// ---- DUTs/IO/PDOs/L1_Current_Status_82DECBF6.TcDUT
{attribute 'GeneratedUsingTerminal: EL3773-0000-0021'}
{attribute addProperty BoxType "EL3773-0000-0021"}
{attribute addProperty Id "I1_StatusAT %I*I1_Status_DC9039207"}
{attribute addProperty CRC "2195639286"}
{attribute addProperty Size "7"}
TYPE L1_Current_Status_82DECBF6 EXTENDS TcoIo.InputBase_8311D824 :
STRUCT
	{attribute addProperty Name "I1_Status"}
	I1_Status AT %I* : I1_Status_DC903920;
END_STRUCT
END_TYPE

// ---- DUTs/IO/PDOs/L1_Current_Samples_9EC08B3E.TcDUT
{attribute 'GeneratedUsingTerminal: EL3773-0000-0021'}
{attribute addProperty BoxType "EL3773-0000-0021"}
{attribute addProperty Id "I1_SamplesAT %I*I1_Samples_2549228720"}
{attribute addProperty CRC "2663418686"}
{attribute addProperty Size "20"}
TYPE L1_Current_Samples_9EC08B3E EXTENDS TcoIo.InputBase_8311D824 :
STRUCT
	{attribute addProperty Name "I1_Samples"}
	I1_Samples AT %I* : I1_Samples_25492287;
END_STRUCT
END_TYPE

// ---- DUTs/IO/PDOs/L2_Voltage_Status_0D1813FE.TcDUT
{attribute 'GeneratedUsingTerminal: EL3773-0000-0021'}
{attribute addProperty BoxType "EL3773-0000-0021"}
{attribute addProperty Id "U2_StatusAT %I*U2_Status_DC9039207"}
{attribute addProperty CRC "219681790"}
{attribute addProperty Size "7"}
TYPE L2_Voltage_Status_0D1813FE EXTENDS TcoIo.InputBase_8311D824 :
STRUCT
	{attribute addProperty Name "U2_Status"}
	U2_Status AT %I* : U2_Status_DC903920;
END_STRUCT
END_TYPE

// ---- DUTs/IO/PDOs/L2_Voltage_Samples_75D833AF.TcDUT
{attribute 'GeneratedUsingTerminal: EL3773-0000-0021'}
{attribute addProperty BoxType "EL3773-0000-0021"}
{attribute addProperty Id "U2_SamplesAT %I*U2_Samples_2549228720"}
{attribute addProperty CRC "1977103279"}
{attribute addProperty Size "20"}
TYPE L2_Voltage_Samples_75D833AF EXTENDS TcoIo.InputBase_8311D824 :
STRUCT
	{attribute addProperty Name "U2_Samples"}
	U2_Samples AT %I* : U2_Samples_25492287;
END_STRUCT
END_TYPE

// ---- DUTs/IO/PDOs/L2_Current_Status_FCB7684B.TcDUT
{attribute 'GeneratedUsingTerminal: EL3773-0000-0021'}
{attribute addProperty BoxType "EL3773-0000-0021"}
{attribute addProperty Id "I2_StatusAT %I*I2_Status_DC9039207"}
{attribute addProperty CRC "4239878219"}
{attribute addProperty Size "7"}
TYPE L2_Current_Status_FCB7684B EXTENDS TcoIo.InputBase_8311D824 :
STRUCT
	{attribute addProperty Name "I2_Status"}
	I2_Status AT %I* : I2_Status_DC903920;
END_STRUCT
END_TYPE

// ---- DUTs/IO/PDOs/L2_Current_Samples_AAB60F6E.TcDUT
{attribute 'GeneratedUsingTerminal: EL3773-0000-0021'}
{attribute addProperty BoxType "EL3773-0000-0021"}
{attribute addProperty Id "I2_SamplesAT %I*I2_Samples_2549228720"}
{attribute addProperty CRC "2864058222"}
{attribute addProperty Size "20"}
TYPE L2_Current_Samples_AAB60F6E EXTENDS TcoIo.InputBase_8311D824 :
STRUCT
	{attribute addProperty Name "I2_Samples"}
	I2_Samples AT %I* : I2_Samples_25492287;
END_STRUCT
END_TYPE

// ---- DUTs/IO/PDOs/L3_Voltage_Status_273F7295.TcDUT
{attribute 'GeneratedUsingTerminal: EL3773-0000-0021'}
{attribute addProperty BoxType "EL3773-0000-0021"}
{attribute addProperty Id "U3_StatusAT %I*U3_Status_DC9039207"}
{attribute addProperty CRC "658469525"}
{attribute addProperty Size "7"}
TYPE L3_Voltage_Status_273F7295 EXTENDS TcoIo.InputBase_8311D824 :
STRUCT
	{attribute addProperty Name "U3_Status"}
	U3_Status AT %I* : U3_Status_DC903920;
END_STRUCT
END_TYPE

// ---- DUTs/IO/PDOs/L3_Voltage_Samples_660A4F9F.TcDUT
{attribute 'GeneratedUsingTerminal: EL3773-0000-0021'}
{attribute addProperty BoxType "EL3773-0000-0021"}
{attribute addProperty Id "U3_SamplesAT %I*U3_Samples_2549228720"}
{attribute addProperty CRC "1711951775"}
{attribute addProperty Size "20"}
TYPE L3_Voltage_Samples_660A4F9F EXTENDS TcoIo.InputBase_8311D824 :
STRUCT
	{attribute addProperty Name "U3_Samples"}
	U3_Samples AT %I* : U3_Samples_25492287;
END_STRUCT
END_TYPE

// ---- DUTs/IO/PDOs/L3_Current_Status_D6900920.TcDUT
{attribute 'GeneratedUsingTerminal: EL3773-0000-0021'}
{attribute addProperty BoxType "EL3773-0000-0021"}
{attribute addProperty Id "I3_StatusAT %I*I3_Status_DC9039207"}
{attribute addProperty CRC "3599763744"}
{attribute addProperty Size "7"}
TYPE L3_Current_Status_D6900920 EXTENDS TcoIo.InputBase_8311D824 :
STRUCT
	{attribute addProperty Name "I3_Status"}
	I3_Status AT %I* : I3_Status_DC903920;
END_STRUCT
END_TYPE

// ---- DUTs/IO/PDOs/L3_Current_Samples_B964735E.TcDUT
{attribute 'GeneratedUsingTerminal: EL3773-0000-0021'}
{attribute addProperty BoxType "EL3773-0000-0021"}
{attribute addProperty Id "I3_SamplesAT %I*I3_Samples_2549228720"}
{attribute addProperty CRC "3110368094"}
{attribute addProperty Size "20"}
TYPE L3_Current_Samples_B964735E EXTENDS TcoIo.InputBase_8311D824 :
STRUCT
	{attribute addProperty Name "I3_Samples"}
	I3_Samples AT %I* : I3_Samples_25492287;
END_STRUCT
END_TYPE

// ---- DUTs/IO/PDOs/AI_NextSync1Time_6DC4D296.TcDUT
{attribute 'GeneratedUsingTerminal: EL3773-0000-0021'}
{attribute addProperty BoxType "EL3773-0000-0021"}
{attribute addProperty Id "StartTimeNextLatchAT %I*StartTimeNextLatch_02E0C1C88"}
{attribute addProperty CRC "1841615510"}
{attribute addProperty Size "8"}
TYPE AI_NextSync1Time_6DC4D296 EXTENDS TcoIo.InputBase_8311D824 :
STRUCT
	{attribute addProperty Name "StartTimeNextLatch"}
	StartTimeNextLatch AT %I* : StartTimeNextLatch_02E0C1C8;
END_STRUCT
END_TYPE

// ---- DUTs/IO/PDOs/AI_Sample_Count_EA88CAD9.TcDUT
{attribute 'GeneratedUsingTerminal: EL3773-0000-0021'}
{attribute addProperty BoxType "EL3773-0000-0021"}
{attribute addProperty Id "Sample_CountAT %I*UINT2"}
{attribute addProperty CRC "3934833369"}
{attribute addProperty Size "2"}
TYPE AI_Sample_Count_EA88CAD9 EXTENDS TcoIo.InputBase_8311D824 :
STRUCT
	{attribute addProperty Name "Sample_Count"}
	Sample_Count AT %I* : UINT;
END_STRUCT
END_TYPE

// ---- DUTs/IO/PDOs/InfoData_B84DBEC5.TcDUT
{attribute 'GeneratedUsingTerminal: EL3773-0000-0021'}
{attribute addProperty BoxType "EL3773-0000-0021"}
{attribute addProperty Id "AdsAddrAT %I*TcoIo.TcoAmsAddr0DcOutputShiftAT %I*DINT4DcInputShiftAT %I*DINT4StateAT %I*UINT2"}
{attribute addProperty CRC "3092102853"}
{attribute addProperty Size "10"}
TYPE InfoData_B84DBEC5 EXTENDS TcoIo.InputBase_8311D824 :
STRUCT
	{attribute addProperty Name "AdsAddr"}
	AdsAddr AT %I* : TcoIo.TcoAmsAddr;
	{attribute addProperty Name "DcOutputShift"}
	DcOutputShift AT %I* : DINT;
	{attribute addProperty Name "DcInputShift"}
	DcInputShift AT %I* : DINT;
	{attribute addProperty Name "State"}
	State AT %I* : UINT;
END_STRUCT
END_TYPE

// ---- DUTs/IO/PDOs/MTO_Inputs_Channel_53C09E8B.TcDUT
{attribute 'GeneratedUsingTerminal: EL2258-0000-0017'}
{attribute addProperty BoxType "EL2258-0000-0017"}
{attribute addProperty Id "StatusAT %I*Status_642C2ED16"}
{attribute addProperty CRC "1405132427"}
{attribute addProperty Size "6"}
TYPE MTO_Inputs_Channel_53C09E8B EXTENDS TcoIo.InputBase_8311D824 :
STRUCT
	{attribute addProperty Name "Status"}
	Status AT %I* : Status_642C2ED1;
END_STRUCT
END_TYPE

// ---- DUTs/IO/PDOs/MTO_Outputs_10x_Channel_A3C0C022.TcDUT
{attribute 'GeneratedUsingTerminal: EL2258-0000-0017'}
{attribute addProperty BoxType "EL2258-0000-0017"}
{attribute addProperty Id "CtrlAT %Q*Ctrl_77460BD36OutputsAT %Q*Outputs_A910484D10Output_event_timeAT %Q*ARRAY[0..9] OF UDINT40"}
{attribute addProperty CRC "922776817"}
{attribute addProperty Size "56"}
TYPE MTO_Outputs_10x_Channel_A3C0C022 EXTENDS TcoIo.OutputBase_10CEE7DE :
STRUCT
	{attribute addProperty Name "Ctrl"}
	Ctrl AT %Q* : Ctrl_77460BD3;
	{attribute addProperty Name "Outputs"}
	Outputs AT %Q* : Outputs_A910484D;
	{attribute addProperty Name "Output_event_time"}
	Output_event_time AT %Q* : ARRAY[0..9] OF UDINT;
END_STRUCT
END_TYPE

// ---- DUTs/IO/PDOs/PM_Inputs_Channel_2F868086.TcDUT
{attribute 'GeneratedUsingTerminal: EL3403-0000-0023'}
{attribute addProperty BoxType "EL3403-0000-0023"}
{attribute addProperty Id "TxPDO_ToggleAT %I*BOOL1CurrentAT %I*DINT4VoltageAT %I*DINT4Active_powerAT %I*DINT4IndexAT %I*USINT1Variant_valueAT %I*DINT4"}
{attribute addProperty CRC "797343878"}
{attribute addProperty Size "18"}
TYPE PM_Inputs_Channel_2F868086 EXTENDS TcoIo.InputBase_8311D824 :
STRUCT
	{attribute addProperty Name "TxPDO_Toggle"}
	TxPDO_Toggle AT %I* : BOOL;
	{attribute addProperty Name "Current"}
	Current AT %I* : DINT;
	{attribute addProperty Name "Voltage"}
	Voltage AT %I* : DINT;
	{attribute addProperty Name "Active_power"}
	Active_power AT %I* : DINT;
	{attribute addProperty Name "Index"}
	Index AT %I* : USINT;
	{attribute addProperty Name "Variant_value"}
	Variant_value AT %I* : DINT;
END_STRUCT
END_TYPE

// ---- DUTs/IO/PDOs/PM_Status_data_2A9514CB.TcDUT
{attribute 'GeneratedUsingTerminal: EL3403-0000-0023'}
{attribute addProperty BoxType "EL3403-0000-0023"}
{attribute addProperty Id "Missing_zero_crossing_AAT %I*BOOL1Missing_zero_crossing_BAT %I*BOOL1Missing_zero_crossing_CAT %I*BOOL1Phase_sequence_errorAT %I*BOOL1"}
{attribute addProperty CRC "714413259"}
{attribute addProperty Size "4"}
TYPE PM_Status_data_2A9514CB EXTENDS TcoIo.InputBase_8311D824 :
STRUCT
	{attribute addProperty Name "Missing_zero_crossing_A"}
	Missing_zero_crossing_A AT %I* : BOOL;
	{attribute addProperty Name "Missing_zero_crossing_B"}
	Missing_zero_crossing_B AT %I* : BOOL;
	{attribute addProperty Name "Missing_zero_crossing_C"}
	Missing_zero_crossing_C AT %I* : BOOL;
	{attribute addProperty Name "Phase_sequence_error"}
	Phase_sequence_error AT %I* : BOOL;
END_STRUCT
END_TYPE

// ---- DUTs/IO/PDOs/PM_Outputs_Channel_E5FBDE30.TcDUT
{attribute 'GeneratedUsingTerminal: EL3403-0000-0023'}
{attribute addProperty BoxType "EL3403-0000-0023"}
{attribute addProperty Id "IndexAT %Q*USINT1"}
{attribute addProperty CRC "3858488880"}
{attribute addProperty Size "1"}
TYPE PM_Outputs_Channel_E5FBDE30 EXTENDS TcoIo.OutputBase_10CEE7DE :
STRUCT
	{attribute addProperty Name "Index"}
	Index AT %Q* : USINT;
END_STRUCT
END_TYPE

// ---- DUTs/IO/PDOs/AT_x_4EC2E768.TcDUT
{attribute 'GeneratedUsingTerminal: AX5101-0000-0214-0214'}
{attribute addProperty BoxType "AX5101-0000-0214-0214"}
{attribute addProperty Id "Drive_status_wordAT %I*UINT2Position_feedback_1_valueAT %I*DINT4Following_distanceAT %I*DINT4"}
{attribute addProperty CRC "1321396072"}
{attribute addProperty Size "10"}
TYPE AT_x_4EC2E768 EXTENDS TcoIo.InputBase_8311D824 :
STRUCT
	{attribute addProperty Name "Drive_status_word"}
	Drive_status_word AT %I* : UINT;
	{attribute addProperty Name "Position_feedback_1_value"}
	Position_feedback_1_value AT %I* : DINT;
	{attribute addProperty Name "Following_distance"}
	Following_distance AT %I* : DINT;
END_STRUCT
END_TYPE

// ---- DUTs/IO/PDOs/MDT_864618EC.TcDUT
{attribute 'GeneratedUsingTerminal: AX5101-0000-0214-0214'}
{attribute addProperty BoxType "AX5101-0000-0214-0214"}
{attribute addProperty Id "Master_control_wordAT %Q*UINT2Position_command_valueAT %Q*DINT4"}
{attribute addProperty CRC "2252740844"}
{attribute addProperty Size "6"}
TYPE MDT_864618EC EXTENDS TcoIo.OutputBase_10CEE7DE :
STRUCT
	{attribute addProperty Name "Master_control_word"}
	Master_control_word AT %Q* : UINT;
	{attribute addProperty Name "Position_command_value"}
	Position_command_value AT %Q* : DINT;
END_STRUCT
END_TYPE

// ---- DUTs/IO/PDOs/InfoData_F60A43AC.TcDUT
{attribute 'GeneratedUsingTerminal: AX5101-0000-0214-0214'}
{attribute addProperty BoxType "AX5101-0000-0214-0214"}
{attribute addProperty Id "AdsAddrAT %I*TcoIo.TcoAmsAddr0DcOutputShiftAT %I*DINT4DcInputShiftAT %I*DINT4Chn0AT %I*USINT1StateAT %I*UINT2"}
{attribute addProperty CRC "4127867820"}
{attribute addProperty Size "11"}
TYPE InfoData_F60A43AC EXTENDS TcoIo.InputBase_8311D824 :
STRUCT
	{attribute addProperty Name "AdsAddr"}
	AdsAddr AT %I* : TcoIo.TcoAmsAddr;
	{attribute addProperty Name "DcOutputShift"}
	DcOutputShift AT %I* : DINT;
	{attribute addProperty Name "DcInputShift"}
	DcInputShift AT %I* : DINT;
	{attribute addProperty Name "Chn0"}
	Chn0 AT %I* : USINT;
	{attribute addProperty Name "State"}
	State AT %I* : UINT;
END_STRUCT
END_TYPE

// ---- DUTs/IO/Boxes/EK1200_013D0B49.TcDUT
{attribute 'GeneratedUsingTerminal: EK1200-1388-0000'}
{attribute addProperty VendorId "#x00000002"}
{attribute addProperty BoxType "EK1200-1388-0000"}
{attribute addProperty Description "EK1200-5000 EtherCAT Power supply (2A E-Bus)"}
{attribute addProperty Physics "YK"}
{attribute addProperty Id "EK1200"}
{attribute addProperty CRC "20777801"}
{attribute addProperty Size "0"}
TYPE EK1200_013D0B49 EXTENDS TcoIo.EtcSlaveBoxBase_77A0E4A7 :
STRUCT
END_STRUCT
END_TYPE

// ---- DUTs/IO/Boxes/EL6002_CD897635.TcDUT
{attribute 'GeneratedUsingTerminal: EL6002-0000-0019'}
{attribute addProperty VendorId "#x00000002"}
{attribute addProperty BoxType "EL6002-0000-0019"}
{attribute addProperty Description "EL6002 Interface 2Ch. (RS232)"}
{attribute addProperty Physics "KK"}
{attribute addProperty Id "COM_TxPDO_Map_Inputs_Channel_1AT %I*COM_TxPDO_Map_Inputs_Channel_3801C95E30COM_TxPDO_Map_Inputs_Channel_2AT %I*COM_TxPDO_Map_Inputs_Channel_3801C95E30COM_RxPDO_Map_Outputs_Channel_1AT %Q*COM_RxPDO_Map_Outputs_Channel_EADA2E0D27COM_RxPDO_Map_Outputs_Channel_2AT %Q*COM_RxPDO_Map_Outputs_Channel_EADA2E0D27WcStateAT %I*WcState_9091E0EB2InfoDataAT %I*InfoData_23CBA8372"}
{attribute addProperty CRC "3448337973"}
{attribute addProperty Size "118"}
TYPE EL6002_CD897635 EXTENDS TcoIo.EtcSlaveTerminalBase_947E5A46 :
STRUCT
	{attribute addProperty Name "COM_TxPDO_Map_Inputs_Channel_1"}
	COM_TxPDO_Map_Inputs_Channel_1 : COM_TxPDO_Map_Inputs_Channel_3801C95E;
	{attribute addProperty Name "COM_TxPDO_Map_Inputs_Channel_2"}
	COM_TxPDO_Map_Inputs_Channel_2 : COM_TxPDO_Map_Inputs_Channel_3801C95E;
	{attribute addProperty Name "COM_RxPDO_Map_Outputs_Channel_1"}
	COM_RxPDO_Map_Outputs_Channel_1 : COM_RxPDO_Map_Outputs_Channel_EADA2E0D;
	{attribute addProperty Name "COM_RxPDO_Map_Outputs_Channel_2"}
	COM_RxPDO_Map_Outputs_Channel_2 : COM_RxPDO_Map_Outputs_Channel_EADA2E0D;
	{attribute addProperty Name "WcState"}
	WcState : TcoIo.WcState_9091E0EB;
	{attribute addProperty Name "InfoData"}
	InfoData : TcoIo.InfoData_23CBA837;
END_STRUCT
END_TYPE

// ---- DUTs/IO/Boxes/EL1809_32157CFD.TcDUT
{attribute 'GeneratedUsingTerminal: EL1809-0000-0018'}
{attribute addProperty VendorId "#x00000002"}
{attribute addProperty BoxType "EL1809-0000-0018"}
{attribute addProperty Description "EL1809 16Ch. Dig. Input 24V, 3ms"}
{attribute addProperty Physics "KK"}
{attribute addProperty Id "Channel_1AT %I*Channel_830843C11Channel_2AT %I*Channel_830843C11Channel_3AT %I*Channel_830843C11Channel_4AT %I*Channel_830843C11Channel_5AT %I*Channel_830843C11Channel_6AT %I*Channel_830843C11Channel_7AT %I*Channel_830843C11Channel_8AT %I*Channel_830843C11Channel_9AT %I*Channel_830843C11Channel_10AT %I*Channel_830843C11Channel_11AT %I*Channel_830843C11Channel_12AT %I*Channel_830843C11Channel_13AT %I*Channel_830843C11Channel_14AT %I*Channel_830843C11Channel_15AT %I*Channel_830843C11Channel_16AT %I*Channel_830843C11WcStateAT %I*WcState_9091E0EB2InfoDataAT %I*InfoData_6F19DB2B2"}
{attribute addProperty CRC "840269053"}
{attribute addProperty Size "20"}
TYPE EL1809_32157CFD EXTENDS TcoIo.EtcSlaveTerminalBase_947E5A46 :
STRUCT
	{attribute addProperty Name "Channel_1"}
	Channel_1 : Channel_830843C1;
	{attribute addProperty Name "Channel_2"}
	Channel_2 : Channel_830843C1;
	{attribute addProperty Name "Channel_3"}
	Channel_3 : Channel_830843C1;
	{attribute addProperty Name "Channel_4"}
	Channel_4 : Channel_830843C1;
	{attribute addProperty Name "Channel_5"}
	Channel_5 : Channel_830843C1;
	{attribute addProperty Name "Channel_6"}
	Channel_6 : Channel_830843C1;
	{attribute addProperty Name "Channel_7"}
	Channel_7 : Channel_830843C1;
	{attribute addProperty Name "Channel_8"}
	Channel_8 : Channel_830843C1;
	{attribute addProperty Name "Channel_9"}
	Channel_9 : Channel_830843C1;
	{attribute addProperty Name "Channel_10"}
	Channel_10 : Channel_830843C1;
	{attribute addProperty Name "Channel_11"}
	Channel_11 : Channel_830843C1;
	{attribute addProperty Name "Channel_12"}
	Channel_12 : Channel_830843C1;
	{attribute addProperty Name "Channel_13"}
	Channel_13 : Channel_830843C1;
	{attribute addProperty Name "Channel_14"}
	Channel_14 : Channel_830843C1;
	{attribute addProperty Name "Channel_15"}
	Channel_15 : Channel_830843C1;
	{attribute addProperty Name "Channel_16"}
	Channel_16 : Channel_830843C1;
	{attribute addProperty Name "WcState"}
	WcState : TcoIo.WcState_9091E0EB;
	{attribute addProperty Name "InfoData"}
	InfoData : TcoIo.InfoData_6F19DB2B;
END_STRUCT
END_TYPE

// ---- DUTs/IO/Boxes/EL2809_2B6483BD.TcDUT
{attribute 'GeneratedUsingTerminal: EL2809-0000-0018'}
{attribute addProperty VendorId "#x00000002"}
{attribute addProperty BoxType "EL2809-0000-0018"}
{attribute addProperty Description "EL2809 16Ch. Dig. Output 24V, 0.5A"}
{attribute addProperty Physics "KK"}
{attribute addProperty Id "Channel_1AT %Q*Channel_42CA91F71Channel_2AT %Q*Channel_42CA91F71Channel_3AT %Q*Channel_42CA91F71Channel_4AT %Q*Channel_42CA91F71Channel_5AT %Q*Channel_42CA91F71Channel_6AT %Q*Channel_42CA91F71Channel_7AT %Q*Channel_42CA91F71Channel_8AT %Q*Channel_42CA91F71Channel_9AT %Q*Channel_42CA91F71Channel_10AT %Q*Channel_42CA91F71Channel_11AT %Q*Channel_42CA91F71Channel_12AT %Q*Channel_42CA91F71Channel_13AT %Q*Channel_42CA91F71Channel_14AT %Q*Channel_42CA91F71Channel_15AT %Q*Channel_42CA91F71Channel_16AT %Q*Channel_42CA91F71WcStateAT %I*WcState_0B2B16F91InfoDataAT %I*InfoData_6F19DB2B2"}
{attribute addProperty CRC "728007613"}
{attribute addProperty Size "19"}
TYPE EL2809_2B6483BD EXTENDS TcoIo.EtcSlaveTerminalBase_947E5A46 :
STRUCT
	{attribute addProperty Name "Channel_1"}
	Channel_1 : Channel_42CA91F7;
	{attribute addProperty Name "Channel_2"}
	Channel_2 : Channel_42CA91F7;
	{attribute addProperty Name "Channel_3"}
	Channel_3 : Channel_42CA91F7;
	{attribute addProperty Name "Channel_4"}
	Channel_4 : Channel_42CA91F7;
	{attribute addProperty Name "Channel_5"}
	Channel_5 : Channel_42CA91F7;
	{attribute addProperty Name "Channel_6"}
	Channel_6 : Channel_42CA91F7;
	{attribute addProperty Name "Channel_7"}
	Channel_7 : Channel_42CA91F7;
	{attribute addProperty Name "Channel_8"}
	Channel_8 : Channel_42CA91F7;
	{attribute addProperty Name "Channel_9"}
	Channel_9 : Channel_42CA91F7;
	{attribute addProperty Name "Channel_10"}
	Channel_10 : Channel_42CA91F7;
	{attribute addProperty Name "Channel_11"}
	Channel_11 : Channel_42CA91F7;
	{attribute addProperty Name "Channel_12"}
	Channel_12 : Channel_42CA91F7;
	{attribute addProperty Name "Channel_13"}
	Channel_13 : Channel_42CA91F7;
	{attribute addProperty Name "Channel_14"}
	Channel_14 : Channel_42CA91F7;
	{attribute addProperty Name "Channel_15"}
	Channel_15 : Channel_42CA91F7;
	{attribute addProperty Name "Channel_16"}
	Channel_16 : Channel_42CA91F7;
	{attribute addProperty Name "WcState"}
	WcState : TcoIo.WcState_0B2B16F9;
	{attribute addProperty Name "InfoData"}
	InfoData : TcoIo.InfoData_6F19DB2B;
END_STRUCT
END_TYPE

// ---- DUTs/IO/Boxes/EL4004_E203F875.TcDUT
{attribute 'GeneratedUsingTerminal: EL4004-0000-0020'}
{attribute addProperty VendorId "#x00000002"}
{attribute addProperty BoxType "EL4004-0000-0020"}
{attribute addProperty Description "EL4004 4Ch. Ana. Output 0-10V, 12bit"}
{attribute addProperty Physics "KK"}
{attribute addProperty Id "AO_Outputs_Channel_1AT %Q*AO_Output_Channel_BA7EBB7C2AO_Outputs_Channel_2AT %Q*AO_Output_Channel_BA7EBB7C2AO_Outputs_Channel_3AT %Q*AO_Output_Channel_BA7EBB7C2AO_Outputs_Channel_4AT %Q*AO_Output_Channel_BA7EBB7C2WcStateAT %I*WcState_0B2B16F91InfoDataAT %I*InfoData_23CBA8372"}
{attribute addProperty CRC "3791911029"}
{attribute addProperty Size "11"}
TYPE EL4004_E203F875 EXTENDS TcoIo.EtcSlaveTerminalBase_947E5A46 :
STRUCT
	{attribute addProperty Name "AO_Outputs_Channel_1"}
	AO_Outputs_Channel_1 : AO_Output_Channel_BA7EBB7C;
	{attribute addProperty Name "AO_Outputs_Channel_2"}
	AO_Outputs_Channel_2 : AO_Output_Channel_BA7EBB7C;
	{attribute addProperty Name "AO_Outputs_Channel_3"}
	AO_Outputs_Channel_3 : AO_Output_Channel_BA7EBB7C;
	{attribute addProperty Name "AO_Outputs_Channel_4"}
	AO_Outputs_Channel_4 : AO_Output_Channel_BA7EBB7C;
	{attribute addProperty Name "WcState"}
	WcState : TcoIo.WcState_0B2B16F9;
	{attribute addProperty Name "InfoData"}
	InfoData : TcoIo.InfoData_23CBA837;
END_STRUCT
END_TYPE

// ---- DUTs/IO/Boxes/EL6001_0DE01E7E.TcDUT
{attribute 'GeneratedUsingTerminal: EL6001-0000-0020'}
{attribute addProperty VendorId "#x00000002"}
{attribute addProperty BoxType "EL6001-0000-0020"}
{attribute addProperty Description "EL6001 Interface (RS232)"}
{attribute addProperty Physics "KK"}
{attribute addProperty Id "COM_InputsAT %I*COM_Inputs_3801C95E30COM_OutputsAT %Q*COM_Outputs_DEF408EC27WcStateAT %I*WcState_9091E0EB2InfoDataAT %I*InfoData_23CBA8372"}
{attribute addProperty CRC "232791678"}
{attribute addProperty Size "61"}
TYPE EL6001_0DE01E7E EXTENDS TcoIo.EtcSlaveTerminalBase_947E5A46 :
STRUCT
	{attribute addProperty Name "COM_Inputs"}
	COM_Inputs : COM_Inputs_3801C95E;
	{attribute addProperty Name "COM_Outputs"}
	COM_Outputs : COM_Outputs_DEF408EC;
	{attribute addProperty Name "WcState"}
	WcState : TcoIo.WcState_9091E0EB;
	{attribute addProperty Name "InfoData"}
	InfoData : TcoIo.InfoData_23CBA837;
END_STRUCT
END_TYPE

// ---- DUTs/IO/Boxes/EL9011_D65D3D32.TcDUT
{attribute 'GeneratedUsingTerminal: EL9011--0000'}
{attribute addProperty VendorId "#x00000002"}
{attribute addProperty BoxType "EL9011--0000"}
{attribute addProperty Description "EL9011 End Terminal"}
{attribute addProperty Physics ""}
{attribute addProperty Id "EL9011"}
{attribute addProperty CRC "3596434738"}
{attribute addProperty Size "0"}
TYPE EL9011_D65D3D32 EXTENDS TcoIo.EtcSlaveEndTerminalBase_866C7F0C :
STRUCT
END_STRUCT
END_TYPE

// ---- DUTs/IO/Boxes/EK1100_1FC0878B.TcDUT
{attribute 'GeneratedUsingTerminal: EK1100-0000-0018'}
{attribute addProperty VendorId "#x00000002"}
{attribute addProperty BoxType "EK1100-0000-0018"}
{attribute addProperty Description "EK1100 EtherCAT Coupler (2A E-Bus)"}
{attribute addProperty Physics "YKY"}
{attribute addProperty Id "InfoDataAT %I*InfoData_6F19DB2B2"}
{attribute addProperty CRC "532711307"}
{attribute addProperty Size "2"}
TYPE EK1100_1FC0878B EXTENDS TcoIo.EtcSlaveBoxBase_77A0E4A7 :
STRUCT
	{attribute addProperty Name "InfoData"}
	InfoData : TcoIo.InfoData_6F19DB2B;
END_STRUCT
END_TYPE

// ---- DUTs/IO/Boxes/EK1122_1FC0878B.TcDUT
{attribute 'GeneratedUsingTerminal: EK1122-0000-0018'}
{attribute addProperty VendorId "#x00000002"}
{attribute addProperty BoxType "EK1122-0000-0018"}
{attribute addProperty Description "EK1122 2 port EtherCAT junction"}
{attribute addProperty Physics "KYKY"}
{attribute addProperty Id "InfoDataAT %I*InfoData_6F19DB2B2"}
{attribute addProperty CRC "532711307"}
{attribute addProperty Size "2"}
TYPE EK1122_1FC0878B EXTENDS TcoIo.EtcSlaveTerminalBase_947E5A46 :
STRUCT
	{attribute addProperty Name "InfoData"}
	InfoData : TcoIo.InfoData_6F19DB2B;
END_STRUCT
END_TYPE

// ---- DUTs/IO/Boxes/EL3174_B71BFF42.TcDUT
{attribute 'GeneratedUsingTerminal: EL3174-0002-0017'}
{attribute addProperty VendorId "#x00000002"}
{attribute addProperty BoxType "EL3174-0002-0017"}
{attribute addProperty Description "EL3174-0002 4Ch. Ana. Input +/-10V, +/-20mA 16 Bit, Isolated Channels"}
{attribute addProperty Physics "KK"}
{attribute addProperty Id "AI_Standard_Channel_1AT %I*AI_Standard_Channel_A8DF64E310AI_Standard_Channel_2AT %I*AI_Standard_Channel_A8DF64E310AI_Standard_Channel_3AT %I*AI_Standard_Channel_A8DF64E310AI_Standard_Channel_4AT %I*AI_Standard_Channel_A8DF64E310WcStateAT %I*WcState_9091E0EB2InfoDataAT %I*InfoData_23CBA8372"}
{attribute addProperty CRC "3072065346"}
{attribute addProperty Size "44"}
TYPE EL3174_B71BFF42 EXTENDS TcoIo.EtcSlaveTerminalBase_947E5A46 :
STRUCT
	{attribute addProperty Name "AI_Standard_Channel_1"}
	AI_Standard_Channel_1 : AI_Standard_Channel_A8DF64E3;
	{attribute addProperty Name "AI_Standard_Channel_2"}
	AI_Standard_Channel_2 : AI_Standard_Channel_A8DF64E3;
	{attribute addProperty Name "AI_Standard_Channel_3"}
	AI_Standard_Channel_3 : AI_Standard_Channel_A8DF64E3;
	{attribute addProperty Name "AI_Standard_Channel_4"}
	AI_Standard_Channel_4 : AI_Standard_Channel_A8DF64E3;
	{attribute addProperty Name "WcState"}
	WcState : TcoIo.WcState_9091E0EB;
	{attribute addProperty Name "InfoData"}
	InfoData : TcoIo.InfoData_23CBA837;
END_STRUCT
END_TYPE

// ---- DUTs/IO/Boxes/EL3011_7A495228.TcDUT
{attribute 'GeneratedUsingTerminal: EL3011-0000-0018'}
{attribute addProperty VendorId "#x00000002"}
{attribute addProperty BoxType "EL3011-0000-0018"}
{attribute addProperty Description "EL3011 4Ch. Ana. Input 0-20mA DIFF"}
{attribute addProperty Physics "KK"}
{attribute addProperty Id "AI_StandardAT %I*AI_Standard_Channel_4A3944819WcStateAT %I*WcState_9091E0EB2InfoDataAT %I*InfoData_23CBA8372"}
{attribute addProperty CRC "2051625512"}
{attribute addProperty Size "13"}
TYPE EL3011_7A495228 EXTENDS TcoIo.EtcSlaveTerminalBase_947E5A46 :
STRUCT
	{attribute addProperty Name "AI_Standard"}
	AI_Standard : AI_Standard_Channel_4A394481;
	{attribute addProperty Name "WcState"}
	WcState : TcoIo.WcState_9091E0EB;
	{attribute addProperty Name "InfoData"}
	InfoData : TcoIo.InfoData_23CBA837;
END_STRUCT
END_TYPE

// ---- DUTs/IO/Boxes/EL2008_E2806B95.TcDUT
{attribute 'GeneratedUsingTerminal: EL2008-0000-0017'}
{attribute addProperty VendorId "#x00000002"}
{attribute addProperty BoxType "EL2008-0000-0017"}
{attribute addProperty Description "EL2008 8Ch. Dig. Output 24V, 0.5A"}
{attribute addProperty Physics "KK"}
{attribute addProperty Id "Channel_1AT %Q*Channel_42CA91F71Channel_2AT %Q*Channel_42CA91F71Channel_3AT %Q*Channel_42CA91F71Channel_4AT %Q*Channel_42CA91F71Channel_5AT %Q*Channel_42CA91F71Channel_6AT %Q*Channel_42CA91F71Channel_7AT %Q*Channel_42CA91F71Channel_8AT %Q*Channel_42CA91F71WcStateAT %I*WcState_0B2B16F91InfoDataAT %I*InfoData_6F19DB2B2"}
{attribute addProperty CRC "3800066965"}
{attribute addProperty Size "11"}
TYPE EL2008_E2806B95 EXTENDS TcoIo.EtcSlaveTerminalBase_947E5A46 :
STRUCT
	{attribute addProperty Name "Channel_1"}
	Channel_1 : Channel_42CA91F7;
	{attribute addProperty Name "Channel_2"}
	Channel_2 : Channel_42CA91F7;
	{attribute addProperty Name "Channel_3"}
	Channel_3 : Channel_42CA91F7;
	{attribute addProperty Name "Channel_4"}
	Channel_4 : Channel_42CA91F7;
	{attribute addProperty Name "Channel_5"}
	Channel_5 : Channel_42CA91F7;
	{attribute addProperty Name "Channel_6"}
	Channel_6 : Channel_42CA91F7;
	{attribute addProperty Name "Channel_7"}
	Channel_7 : Channel_42CA91F7;
	{attribute addProperty Name "Channel_8"}
	Channel_8 : Channel_42CA91F7;
	{attribute addProperty Name "WcState"}
	WcState : TcoIo.WcState_0B2B16F9;
	{attribute addProperty Name "InfoData"}
	InfoData : TcoIo.InfoData_6F19DB2B;
END_STRUCT
END_TYPE

// ---- DUTs/IO/Boxes/EK1110_1FC0878B.TcDUT
{attribute 'GeneratedUsingTerminal: EK1110-0000-0017'}
{attribute addProperty VendorId "#x00000002"}
{attribute addProperty BoxType "EK1110-0000-0017"}
{attribute addProperty Description "EK1110 EtherCAT extension"}
{attribute addProperty Physics "KY"}
{attribute addProperty Id "InfoDataAT %I*InfoData_6F19DB2B2"}
{attribute addProperty CRC "532711307"}
{attribute addProperty Size "2"}
TYPE EK1110_1FC0878B EXTENDS TcoIo.EtcSlaveTerminalBase_947E5A46 :
STRUCT
	{attribute addProperty Name "InfoData"}
	InfoData : TcoIo.InfoData_6F19DB2B;
END_STRUCT
END_TYPE

// ---- DUTs/IO/Boxes/EL1819_32157CFD.TcDUT
{attribute 'GeneratedUsingTerminal: EL1819-0000-0018'}
{attribute addProperty VendorId "#x00000002"}
{attribute addProperty BoxType "EL1819-0000-0018"}
{attribute addProperty Description "EL1819 16Ch. Dig. Input 24V, 10Ã‚Âµs"}
{attribute addProperty Physics "KK"}
{attribute addProperty Id "Channel_1AT %I*Channel_830843C11Channel_2AT %I*Channel_830843C11Channel_3AT %I*Channel_830843C11Channel_4AT %I*Channel_830843C11Channel_5AT %I*Channel_830843C11Channel_6AT %I*Channel_830843C11Channel_7AT %I*Channel_830843C11Channel_8AT %I*Channel_830843C11Channel_9AT %I*Channel_830843C11Channel_10AT %I*Channel_830843C11Channel_11AT %I*Channel_830843C11Channel_12AT %I*Channel_830843C11Channel_13AT %I*Channel_830843C11Channel_14AT %I*Channel_830843C11Channel_15AT %I*Channel_830843C11Channel_16AT %I*Channel_830843C11WcStateAT %I*WcState_9091E0EB2InfoDataAT %I*InfoData_6F19DB2B2"}
{attribute addProperty CRC "840269053"}
{attribute addProperty Size "20"}
TYPE EL1819_32157CFD EXTENDS TcoIo.EtcSlaveTerminalBase_947E5A46 :
STRUCT
	{attribute addProperty Name "Channel_1"}
	Channel_1 : Channel_830843C1;
	{attribute addProperty Name "Channel_2"}
	Channel_2 : Channel_830843C1;
	{attribute addProperty Name "Channel_3"}
	Channel_3 : Channel_830843C1;
	{attribute addProperty Name "Channel_4"}
	Channel_4 : Channel_830843C1;
	{attribute addProperty Name "Channel_5"}
	Channel_5 : Channel_830843C1;
	{attribute addProperty Name "Channel_6"}
	Channel_6 : Channel_830843C1;
	{attribute addProperty Name "Channel_7"}
	Channel_7 : Channel_830843C1;
	{attribute addProperty Name "Channel_8"}
	Channel_8 : Channel_830843C1;
	{attribute addProperty Name "Channel_9"}
	Channel_9 : Channel_830843C1;
	{attribute addProperty Name "Channel_10"}
	Channel_10 : Channel_830843C1;
	{attribute addProperty Name "Channel_11"}
	Channel_11 : Channel_830843C1;
	{attribute addProperty Name "Channel_12"}
	Channel_12 : Channel_830843C1;
	{attribute addProperty Name "Channel_13"}
	Channel_13 : Channel_830843C1;
	{attribute addProperty Name "Channel_14"}
	Channel_14 : Channel_830843C1;
	{attribute addProperty Name "Channel_15"}
	Channel_15 : Channel_830843C1;
	{attribute addProperty Name "Channel_16"}
	Channel_16 : Channel_830843C1;
	{attribute addProperty Name "WcState"}
	WcState : TcoIo.WcState_9091E0EB;
	{attribute addProperty Name "InfoData"}
	InfoData : TcoIo.InfoData_6F19DB2B;
END_STRUCT
END_TYPE

// ---- DUTs/IO/Boxes/EL2788_E2806B95.TcDUT
{attribute 'GeneratedUsingTerminal: EL2788-0000-0016'}
{attribute addProperty VendorId "#x00000002"}
{attribute addProperty BoxType "EL2788-0000-0016"}
{attribute addProperty Description "EL2788 8Ch. Dig. Output 24V AC/DC, 2A"}
{attribute addProperty Physics "KK"}
{attribute addProperty Id "Channel_1AT %Q*Channel_42CA91F71Channel_2AT %Q*Channel_42CA91F71Channel_3AT %Q*Channel_42CA91F71Channel_4AT %Q*Channel_42CA91F71Channel_5AT %Q*Channel_42CA91F71Channel_6AT %Q*Channel_42CA91F71Channel_7AT %Q*Channel_42CA91F71Channel_8AT %Q*Channel_42CA91F71WcStateAT %I*WcState_0B2B16F91InfoDataAT %I*InfoData_6F19DB2B2"}
{attribute addProperty CRC "3800066965"}
{attribute addProperty Size "11"}
TYPE EL2788_E2806B95 EXTENDS TcoIo.EtcSlaveTerminalBase_947E5A46 :
STRUCT
	{attribute addProperty Name "Channel_1"}
	Channel_1 : Channel_42CA91F7;
	{attribute addProperty Name "Channel_2"}
	Channel_2 : Channel_42CA91F7;
	{attribute addProperty Name "Channel_3"}
	Channel_3 : Channel_42CA91F7;
	{attribute addProperty Name "Channel_4"}
	Channel_4 : Channel_42CA91F7;
	{attribute addProperty Name "Channel_5"}
	Channel_5 : Channel_42CA91F7;
	{attribute addProperty Name "Channel_6"}
	Channel_6 : Channel_42CA91F7;
	{attribute addProperty Name "Channel_7"}
	Channel_7 : Channel_42CA91F7;
	{attribute addProperty Name "Channel_8"}
	Channel_8 : Channel_42CA91F7;
	{attribute addProperty Name "WcState"}
	WcState : TcoIo.WcState_0B2B16F9;
	{attribute addProperty Name "InfoData"}
	InfoData : TcoIo.InfoData_6F19DB2B;
END_STRUCT
END_TYPE

// ---- DUTs/IO/Boxes/EL3773_F128CC82.TcDUT
{attribute 'GeneratedUsingTerminal: EL3773-0000-0021'}
{attribute addProperty VendorId "#x00000002"}
{attribute addProperty BoxType "EL3773-0000-0021"}
{attribute addProperty Description "EL3773 3 Ch. Power Monitoring, Oversample"}
{attribute addProperty Physics "KK"}
{attribute addProperty Id "L1_Voltage_StatusAT %I*L1_Voltage_Status_7371B0437L1_Voltage_SamplesAT %I*L1_Voltage_Samples_41AEB7FF20L1_Current_StatusAT %I*L1_Current_Status_82DECBF67L1_Current_SamplesAT %I*L1_Current_Samples_9EC08B3E20L2_Voltage_StatusAT %I*L2_Voltage_Status_0D1813FE7L2_Voltage_SamplesAT %I*L2_Voltage_Samples_75D833AF20L2_Current_StatusAT %I*L2_Current_Status_FCB7684B7L2_Current_SamplesAT %I*L2_Current_Samples_AAB60F6E20L3_Voltage_StatusAT %I*L3_Voltage_Status_273F72957L3_Voltage_SamplesAT %I*L3_Voltage_Samples_660A4F9F20L3_Current_StatusAT %I*L3_Current_Status_D69009207L3_Current_SamplesAT %I*L3_Current_Samples_B964735E20AI_NextSync1TimeAT %I*AI_NextSync1Time_6DC4D2968AI_Sample_CountAT %I*AI_Sample_Count_EA88CAD92WcStateAT %I*WcState_9091E0EB2InfoDataAT %I*InfoData_B84DBEC510"}
{attribute addProperty CRC "4045982850"}
{attribute addProperty Size "184"}
TYPE EL3773_F128CC82 EXTENDS TcoIo.EtcSlaveTerminalBase_947E5A46 :
STRUCT
	{attribute addProperty Name "L1_Voltage_Status"}
	L1_Voltage_Status : L1_Voltage_Status_7371B043;
	{attribute addProperty Name "L1_Voltage_Samples"}
	L1_Voltage_Samples : L1_Voltage_Samples_41AEB7FF;
	{attribute addProperty Name "L1_Current_Status"}
	L1_Current_Status : L1_Current_Status_82DECBF6;
	{attribute addProperty Name "L1_Current_Samples"}
	L1_Current_Samples : L1_Current_Samples_9EC08B3E;
	{attribute addProperty Name "L2_Voltage_Status"}
	L2_Voltage_Status : L2_Voltage_Status_0D1813FE;
	{attribute addProperty Name "L2_Voltage_Samples"}
	L2_Voltage_Samples : L2_Voltage_Samples_75D833AF;
	{attribute addProperty Name "L2_Current_Status"}
	L2_Current_Status : L2_Current_Status_FCB7684B;
	{attribute addProperty Name "L2_Current_Samples"}
	L2_Current_Samples : L2_Current_Samples_AAB60F6E;
	{attribute addProperty Name "L3_Voltage_Status"}
	L3_Voltage_Status : L3_Voltage_Status_273F7295;
	{attribute addProperty Name "L3_Voltage_Samples"}
	L3_Voltage_Samples : L3_Voltage_Samples_660A4F9F;
	{attribute addProperty Name "L3_Current_Status"}
	L3_Current_Status : L3_Current_Status_D6900920;
	{attribute addProperty Name "L3_Current_Samples"}
	L3_Current_Samples : L3_Current_Samples_B964735E;
	{attribute addProperty Name "AI_NextSync1Time"}
	AI_NextSync1Time : AI_NextSync1Time_6DC4D296;
	{attribute addProperty Name "AI_Sample_Count"}
	AI_Sample_Count : AI_Sample_Count_EA88CAD9;
	{attribute addProperty Name "WcState"}
	WcState : TcoIo.WcState_9091E0EB;
	{attribute addProperty Name "InfoData"}
	InfoData : InfoData_B84DBEC5;
END_STRUCT
END_TYPE

// ---- DUTs/IO/Boxes/EL2258_E3B260FA.TcDUT
{attribute 'GeneratedUsingTerminal: EL2258-0000-0017'}
{attribute addProperty VendorId "#x00000002"}
{attribute addProperty BoxType "EL2258-0000-0017"}
{attribute addProperty Description "EL2258 8Ch. Dig Output 24V with Multi-Time-Stamp"}
{attribute addProperty Physics "KK"}
{attribute addProperty Id "MTO_Inputs_Channel_1AT %I*MTO_Inputs_Channel_53C09E8B6MTO_Inputs_Channel_2AT %I*MTO_Inputs_Channel_53C09E8B6MTO_Inputs_Channel_3AT %I*MTO_Inputs_Channel_53C09E8B6MTO_Inputs_Channel_4AT %I*MTO_Inputs_Channel_53C09E8B6MTO_Inputs_Channel_5AT %I*MTO_Inputs_Channel_53C09E8B6MTO_Inputs_Channel_6AT %I*MTO_Inputs_Channel_53C09E8B6MTO_Inputs_Channel_7AT %I*MTO_Inputs_Channel_53C09E8B6MTO_Inputs_Channel_8AT %I*MTO_Inputs_Channel_53C09E8B6MTO_Outputs_10x_Channel_1AT %Q*MTO_Outputs_10x_Channel_A3C0C02256MTO_Outputs_10x_Channel_2AT %Q*MTO_Outputs_10x_Channel_A3C0C02256MTO_Outputs_10x_Channel_3AT %Q*MTO_Outputs_10x_Channel_A3C0C02256MTO_Outputs_10x_Channel_4AT %Q*MTO_Outputs_10x_Channel_A3C0C02256MTO_Outputs_10x_Channel_5AT %Q*MTO_Outputs_10x_Channel_A3C0C02256MTO_Outputs_10x_Channel_6AT %Q*MTO_Outputs_10x_Channel_A3C0C02256MTO_Outputs_10x_Channel_7AT %Q*MTO_Outputs_10x_Channel_A3C0C02256MTO_Outputs_10x_Channel_8AT %Q*MTO_Outputs_10x_Channel_A3C0C02256WcStateAT %I*WcState_9091E0EB2InfoDataAT %I*InfoData_B84DBEC510"}
{attribute addProperty CRC "3820118266"}
{attribute addProperty Size "508"}
TYPE EL2258_E3B260FA EXTENDS TcoIo.EtcSlaveTerminalBase_947E5A46 :
STRUCT
	{attribute addProperty Name "MTO_Inputs_Channel_1"}
	MTO_Inputs_Channel_1 : MTO_Inputs_Channel_53C09E8B;
	{attribute addProperty Name "MTO_Inputs_Channel_2"}
	MTO_Inputs_Channel_2 : MTO_Inputs_Channel_53C09E8B;
	{attribute addProperty Name "MTO_Inputs_Channel_3"}
	MTO_Inputs_Channel_3 : MTO_Inputs_Channel_53C09E8B;
	{attribute addProperty Name "MTO_Inputs_Channel_4"}
	MTO_Inputs_Channel_4 : MTO_Inputs_Channel_53C09E8B;
	{attribute addProperty Name "MTO_Inputs_Channel_5"}
	MTO_Inputs_Channel_5 : MTO_Inputs_Channel_53C09E8B;
	{attribute addProperty Name "MTO_Inputs_Channel_6"}
	MTO_Inputs_Channel_6 : MTO_Inputs_Channel_53C09E8B;
	{attribute addProperty Name "MTO_Inputs_Channel_7"}
	MTO_Inputs_Channel_7 : MTO_Inputs_Channel_53C09E8B;
	{attribute addProperty Name "MTO_Inputs_Channel_8"}
	MTO_Inputs_Channel_8 : MTO_Inputs_Channel_53C09E8B;
	{attribute addProperty Name "MTO_Outputs_10x_Channel_1"}
	MTO_Outputs_10x_Channel_1 : MTO_Outputs_10x_Channel_A3C0C022;
	{attribute addProperty Name "MTO_Outputs_10x_Channel_2"}
	MTO_Outputs_10x_Channel_2 : MTO_Outputs_10x_Channel_A3C0C022;
	{attribute addProperty Name "MTO_Outputs_10x_Channel_3"}
	MTO_Outputs_10x_Channel_3 : MTO_Outputs_10x_Channel_A3C0C022;
	{attribute addProperty Name "MTO_Outputs_10x_Channel_4"}
	MTO_Outputs_10x_Channel_4 : MTO_Outputs_10x_Channel_A3C0C022;
	{attribute addProperty Name "MTO_Outputs_10x_Channel_5"}
	MTO_Outputs_10x_Channel_5 : MTO_Outputs_10x_Channel_A3C0C022;
	{attribute addProperty Name "MTO_Outputs_10x_Channel_6"}
	MTO_Outputs_10x_Channel_6 : MTO_Outputs_10x_Channel_A3C0C022;
	{attribute addProperty Name "MTO_Outputs_10x_Channel_7"}
	MTO_Outputs_10x_Channel_7 : MTO_Outputs_10x_Channel_A3C0C022;
	{attribute addProperty Name "MTO_Outputs_10x_Channel_8"}
	MTO_Outputs_10x_Channel_8 : MTO_Outputs_10x_Channel_A3C0C022;
	{attribute addProperty Name "WcState"}
	WcState : TcoIo.WcState_9091E0EB;
	{attribute addProperty Name "InfoData"}
	InfoData : InfoData_B84DBEC5;
END_STRUCT
END_TYPE

// ---- DUTs/IO/Boxes/EL3164_B71BFF42.TcDUT
{attribute 'GeneratedUsingTerminal: EL3164-0000-0020'}
{attribute addProperty VendorId "#x00000002"}
{attribute addProperty BoxType "EL3164-0000-0020"}
{attribute addProperty Description "EL3164 4Ch. Ana. Input 0-10V"}
{attribute addProperty Physics "KK"}
{attribute addProperty Id "AI_Standard_Channel_1AT %I*AI_Standard_Channel_A8DF64E310AI_Standard_Channel_2AT %I*AI_Standard_Channel_A8DF64E310AI_Standard_Channel_3AT %I*AI_Standard_Channel_A8DF64E310AI_Standard_Channel_4AT %I*AI_Standard_Channel_A8DF64E310WcStateAT %I*WcState_9091E0EB2InfoDataAT %I*InfoData_23CBA8372"}
{attribute addProperty CRC "3072065346"}
{attribute addProperty Size "44"}
TYPE EL3164_B71BFF42 EXTENDS TcoIo.EtcSlaveTerminalBase_947E5A46 :
STRUCT
	{attribute addProperty Name "AI_Standard_Channel_1"}
	AI_Standard_Channel_1 : AI_Standard_Channel_A8DF64E3;
	{attribute addProperty Name "AI_Standard_Channel_2"}
	AI_Standard_Channel_2 : AI_Standard_Channel_A8DF64E3;
	{attribute addProperty Name "AI_Standard_Channel_3"}
	AI_Standard_Channel_3 : AI_Standard_Channel_A8DF64E3;
	{attribute addProperty Name "AI_Standard_Channel_4"}
	AI_Standard_Channel_4 : AI_Standard_Channel_A8DF64E3;
	{attribute addProperty Name "WcState"}
	WcState : TcoIo.WcState_9091E0EB;
	{attribute addProperty Name "InfoData"}
	InfoData : TcoIo.InfoData_23CBA837;
END_STRUCT
END_TYPE

// ---- DUTs/IO/Boxes/EL1008_78E8D3DD.TcDUT
{attribute 'GeneratedUsingTerminal: EL1008-0000-0018'}
{attribute addProperty VendorId "#x00000002"}
{attribute addProperty BoxType "EL1008-0000-0018"}
{attribute addProperty Description "EL1008 8Ch. Dig. Input 24V, 3ms"}
{attribute addProperty Physics "KK"}
{attribute addProperty Id "Channel_1AT %I*Channel_830843C11Channel_2AT %I*Channel_830843C11Channel_3AT %I*Channel_830843C11Channel_4AT %I*Channel_830843C11Channel_5AT %I*Channel_830843C11Channel_6AT %I*Channel_830843C11Channel_7AT %I*Channel_830843C11Channel_8AT %I*Channel_830843C11WcStateAT %I*WcState_9091E0EB2InfoDataAT %I*InfoData_6F19DB2B2"}
{attribute addProperty CRC "2028524509"}
{attribute addProperty Size "12"}
TYPE EL1008_78E8D3DD EXTENDS TcoIo.EtcSlaveTerminalBase_947E5A46 :
STRUCT
	{attribute addProperty Name "Channel_1"}
	Channel_1 : Channel_830843C1;
	{attribute addProperty Name "Channel_2"}
	Channel_2 : Channel_830843C1;
	{attribute addProperty Name "Channel_3"}
	Channel_3 : Channel_830843C1;
	{attribute addProperty Name "Channel_4"}
	Channel_4 : Channel_830843C1;
	{attribute addProperty Name "Channel_5"}
	Channel_5 : Channel_830843C1;
	{attribute addProperty Name "Channel_6"}
	Channel_6 : Channel_830843C1;
	{attribute addProperty Name "Channel_7"}
	Channel_7 : Channel_830843C1;
	{attribute addProperty Name "Channel_8"}
	Channel_8 : Channel_830843C1;
	{attribute addProperty Name "WcState"}
	WcState : TcoIo.WcState_9091E0EB;
	{attribute addProperty Name "InfoData"}
	InfoData : TcoIo.InfoData_6F19DB2B;
END_STRUCT
END_TYPE

// ---- DUTs/IO/Boxes/EL3403_812980A6.TcDUT
{attribute 'GeneratedUsingTerminal: EL3403-0000-0023'}
{attribute addProperty VendorId "#x00000002"}
{attribute addProperty BoxType "EL3403-0000-0023"}
{attribute addProperty Description "EL3403 3Ch. Power Measuring"}
{attribute addProperty Physics "KK"}
{attribute addProperty Id "PM_Inputs_Channel_1AT %I*PM_Inputs_Channel_2F86808618PM_Inputs_Channel_2AT %I*PM_Inputs_Channel_2F86808618PM_Inputs_Channel_3AT %I*PM_Inputs_Channel_2F86808618PM_Status_dataAT %I*PM_Status_data_2A9514CB4PM_Outputs_Channel_1AT %Q*PM_Outputs_Channel_E5FBDE301PM_Outputs_Channel_2AT %Q*PM_Outputs_Channel_E5FBDE301PM_Outputs_Channel_3AT %Q*PM_Outputs_Channel_E5FBDE301WcStateAT %I*WcState_9091E0EB2InfoDataAT %I*InfoData_23CBA8372"}
{attribute addProperty CRC "2166980774"}
{attribute addProperty Size "65"}
TYPE EL3403_812980A6 EXTENDS TcoIo.EtcSlaveTerminalBase_947E5A46 :
STRUCT
	{attribute addProperty Name "PM_Inputs_Channel_1"}
	PM_Inputs_Channel_1 : PM_Inputs_Channel_2F868086;
	{attribute addProperty Name "PM_Inputs_Channel_2"}
	PM_Inputs_Channel_2 : PM_Inputs_Channel_2F868086;
	{attribute addProperty Name "PM_Inputs_Channel_3"}
	PM_Inputs_Channel_3 : PM_Inputs_Channel_2F868086;
	{attribute addProperty Name "PM_Status_data"}
	PM_Status_data : PM_Status_data_2A9514CB;
	{attribute addProperty Name "PM_Outputs_Channel_1"}
	PM_Outputs_Channel_1 : PM_Outputs_Channel_E5FBDE30;
	{attribute addProperty Name "PM_Outputs_Channel_2"}
	PM_Outputs_Channel_2 : PM_Outputs_Channel_E5FBDE30;
	{attribute addProperty Name "PM_Outputs_Channel_3"}
	PM_Outputs_Channel_3 : PM_Outputs_Channel_E5FBDE30;
	{attribute addProperty Name "WcState"}
	WcState : TcoIo.WcState_9091E0EB;
	{attribute addProperty Name "InfoData"}
	InfoData : TcoIo.InfoData_23CBA837;
END_STRUCT
END_TYPE

// ---- DUTs/IO/Boxes/EL3024_C6E76B5A.TcDUT
{attribute 'GeneratedUsingTerminal: EL3024-0000-0018'}
{attribute addProperty VendorId "#x00000002"}
{attribute addProperty BoxType "EL3024-0000-0018"}
{attribute addProperty Description "EL3024 4Ch. Ana. Input 4-20mA DIFF"}
{attribute addProperty Physics "KK"}
{attribute addProperty Id "AI_Standard_Channel_1AT %I*AI_Standard_Channel_4A3944819AI_Standard_Channel_2AT %I*AI_Standard_Channel_4A3944819AI_Standard_Channel_3AT %I*AI_Standard_Channel_4A3944819AI_Standard_Channel_4AT %I*AI_Standard_Channel_4A3944819WcStateAT %I*WcState_9091E0EB2InfoDataAT %I*InfoData_23CBA8372"}
{attribute addProperty CRC "3337055066"}
{attribute addProperty Size "40"}
TYPE EL3024_C6E76B5A EXTENDS TcoIo.EtcSlaveTerminalBase_947E5A46 :
STRUCT
	{attribute addProperty Name "AI_Standard_Channel_1"}
	AI_Standard_Channel_1 : AI_Standard_Channel_4A394481;
	{attribute addProperty Name "AI_Standard_Channel_2"}
	AI_Standard_Channel_2 : AI_Standard_Channel_4A394481;
	{attribute addProperty Name "AI_Standard_Channel_3"}
	AI_Standard_Channel_3 : AI_Standard_Channel_4A394481;
	{attribute addProperty Name "AI_Standard_Channel_4"}
	AI_Standard_Channel_4 : AI_Standard_Channel_4A394481;
	{attribute addProperty Name "WcState"}
	WcState : TcoIo.WcState_9091E0EB;
	{attribute addProperty Name "InfoData"}
	InfoData : TcoIo.InfoData_23CBA837;
END_STRUCT
END_TYPE

// ---- DUTs/IO/Boxes/AX5101_1BD22F51.TcDUT
{attribute 'GeneratedUsingTerminal: AX5101-0000-0214-0214'}
{attribute addProperty VendorId "#x00000002"}
{attribute addProperty BoxType "AX5101-0000-0214-0214"}
{attribute addProperty Description "AX5101-0000-0214 EtherCAT Drive (SoE, 1 Ch.)"}
{attribute addProperty Physics "YY_K"}
{attribute addProperty Id "AT_xAT %I*AT_x_4EC2E76810MDTAT %Q*MDT_864618EC6WcStateAT %I*WcState_9091E0EB2InfoDataAT %I*InfoData_F60A43AC11"}
{attribute addProperty CRC "466759505"}
{attribute addProperty Size "29"}
TYPE AX5101_1BD22F51 EXTENDS TcoIo.EtcSlaveBoxBase_77A0E4A7 :
STRUCT
	{attribute addProperty Name "AT_x"}
	AT_x : AT_x_4EC2E768;
	{attribute addProperty Name "MDT"}
	MDT : MDT_864618EC;
	{attribute addProperty Name "WcState"}
	WcState : TcoIo.WcState_9091E0EB;
	{attribute addProperty Name "InfoData"}
	InfoData : InfoData_F60A43AC;
END_STRUCT
END_TYPE

// ---- DUTs/IO/Devices/SyncUnitTasks_4BE01469.TcDUT
{attribute 'GeneratedUsingTerminal: '}
{attribute addProperty BoxType ""}
{attribute addProperty Id "unreferencedAT %I*SyncUnitTask_AB2F50799PlcTaskAT %I*SyncUnitTask_AB2F50799"}
{attribute addProperty CRC "1272976489"}
{attribute addProperty Size "18"}
TYPE SyncUnitTasks_4BE01469 EXTENDS TcoIo.SyncUnitTasksBase_7C8711EB :
STRUCT
	{attribute addProperty Name "unreferenced"}
	unreferenced : TcoIo.SyncUnitTask_AB2F5079;
	{attribute addProperty Name "PlcTask"}
	PlcTask : TcoIo.SyncUnitTask_AB2F5079;
END_STRUCT
END_TYPE

// ---- DUTs/IO/Devices/SyncUnits_67D36DDA.TcDUT
{attribute 'GeneratedUsingTerminal: '}
{attribute addProperty BoxType ""}
{attribute addProperty Id "_defaultAT %I*SyncUnitTasks_4BE0146918"}
{attribute addProperty CRC "1741909466"}
{attribute addProperty Size "18"}
TYPE SyncUnits_67D36DDA EXTENDS TcoIo.SyncUnitsBase_AD6C35CE :
STRUCT
	{attribute addProperty Name "_default"}
	_default : SyncUnitTasks_4BE01469;
END_STRUCT
END_TYPE

// ---- DUTs/IO/Devices/SyncUnits_91A42BBF.TcDUT
{attribute 'GeneratedUsingTerminal: '}
{attribute addProperty BoxType ""}
{attribute addProperty Id "_defaultAT %I*SyncUnitTasks_4BE0146918Row_0AT %I*SyncUnitTasks_4BE0146918Row_1AT %I*SyncUnitTasks_4BE0146918Row_2AT %I*SyncUnitTasks_4BE0146918Row_3AT %I*SyncUnitTasks_4BE0146918Row_4AT %I*SyncUnitTasks_4BE0146918"}
{attribute addProperty CRC "2443455423"}
{attribute addProperty Size "108"}
TYPE SyncUnits_91A42BBF EXTENDS TcoIo.SyncUnitsBase_AD6C35CE :
STRUCT
	{attribute addProperty Name "_default"}
	_default : SyncUnitTasks_4BE01469;
	{attribute addProperty Name "Row_0"}
	Row_0 : SyncUnitTasks_4BE01469;
	{attribute addProperty Name "Row_1"}
	Row_1 : SyncUnitTasks_4BE01469;
	{attribute addProperty Name "Row_2"}
	Row_2 : SyncUnitTasks_4BE01469;
	{attribute addProperty Name "Row_3"}
	Row_3 : SyncUnitTasks_4BE01469;
	{attribute addProperty Name "Row_4"}
	Row_4 : SyncUnitTasks_4BE01469;
END_STRUCT
END_TYPE

// ---- DUTs/IO/Topology/Term_1_EK1200_B38DC9A8.TcDUT
{attribute 'GeneratedUsingTerminal: EK1200-1388-0000'}
{attribute addProperty BoxType "EK1200-1388-0000"}
{attribute addProperty Id "Term_2_EL6002EL6002_CD897635118Term_3_EL1809EL1809_32157CFD20Term_4_EL2809EL2809_2B6483BD19Term_5_EL4004EL4004_E203F87511Term_6_EL2809EL2809_2B6483BD19Term_7_EL6001EL6001_0DE01E7E61Term_8_EL9011EL9011_D65D3D320"}
{attribute addProperty CRC "3012413864"}
{attribute addProperty Size "248"}
{attribute addProperty Name "Term 1 (EK1200)"}
TYPE Term_1_EK1200_B38DC9A8 EXTENDS EK1200_013D0B49 :
STRUCT
	{attribute addProperty Name "Term 2 (EL6002)"}
	{attribute addProperty PreviousPort "Term 1 (EK1200) : B"}
	{attribute addProperty SyncUnit "default"}
	Term_2_EL6002 : EL6002_CD897635;
	{attribute addProperty Name "Term 3 (EL1809)"}
	{attribute addProperty PreviousPort "Term 2 (EL6002) : B"}
	{attribute addProperty SyncUnit "default"}
	Term_3_EL1809 : EL1809_32157CFD;
	{attribute addProperty Name "Term 4 (EL2809)"}
	{attribute addProperty PreviousPort "Term 3 (EL1809) : B"}
	{attribute addProperty SyncUnit "default"}
	Term_4_EL2809 : EL2809_2B6483BD;
	{attribute addProperty Name "Term 5 (EL4004)"}
	{attribute addProperty PreviousPort "Term 4 (EL2809) : B"}
	{attribute addProperty SyncUnit "default"}
	Term_5_EL4004 : EL4004_E203F875;
	{attribute addProperty Name "Term 6 (EL2809)"}
	{attribute addProperty PreviousPort "Term 5 (EL4004) : B"}
	{attribute addProperty SyncUnit "default"}
	Term_6_EL2809 : EL2809_2B6483BD;
	{attribute addProperty Name "Term 7 (EL6001)"}
	{attribute addProperty PreviousPort "Term 6 (EL2809) : B"}
	{attribute addProperty SyncUnit "default"}
	Term_7_EL6001 : EL6001_0DE01E7E;
	{attribute addProperty Name "Term 8 (EL9011)"}
	{attribute addProperty PreviousPort "Term 7 (EL6001) : B"}
	{attribute addProperty SyncUnit "default"}
	Term_8_EL9011 : EL9011_D65D3D32;
END_STRUCT
END_TYPE

// ---- DUTs/IO/Topology/Device_1_EtherCAT_B557D6C6.TcDUT
{attribute 'GeneratedUsingTerminal: IODEVICETYPE_ETHERCATPROT'}
{attribute addProperty BoxType "IODEVICETYPE_ETHERCATPROT"}
{attribute addProperty Id "Term_1_EK1200Term_1_EK1200_B38DC9A8248SyncUnitsSyncUnits_67D36DDA18InputsInputs_A65FACA410OutputsOutputs_23C0ED1D6InfoDataInfoData_84133AC922"}
{attribute addProperty CRC "3042432710"}
{attribute addProperty Size "304"}
{attribute addProperty Name "Device 1 (EtherCAT)"}
TYPE Device_1_EtherCAT_B557D6C6 EXTENDS TcoIo.EtcMasterBase_62654B43 :
STRUCT
	{attribute addProperty Name "Term 1 (EK1200)"}
	{attribute addProperty PreviousPort "Device 1 (EtherCAT) : Master"}
	{attribute addProperty SyncUnit "default"}
	Term_1_EK1200 : Term_1_EK1200_B38DC9A8;
	{attribute addProperty Name "SyncUnits"}
	SyncUnits : SyncUnits_67D36DDA;
	{attribute addProperty Name "Inputs"}
	Inputs : TcoIo.Inputs_A65FACA4;
	{attribute addProperty Name "Outputs"}
	Outputs : TcoIo.Outputs_23C0ED1D;
	{attribute addProperty Name "InfoData"}
	InfoData : TcoIo.InfoData_84133AC9;
END_STRUCT
END_TYPE

// ---- DUTs/IO/Topology/Term_11_EK1100_B6553301.TcDUT
{attribute 'GeneratedUsingTerminal: EK1100-0000-0018'}
{attribute addProperty BoxType "EK1100-0000-0018"}
{attribute addProperty Id "Term_12_EL3174_0002EL3174_B71BFF4244Term_13_EL6001EL6001_0DE01E7E61Term_14_EL3011EL3011_7A49522813Term_15_EL2008EL2008_E2806B9511Term_16_EL2008EL2008_E2806B9511Term_17_EK1110EK1110_1FC0878B2"}
{attribute addProperty CRC "3059036929"}
{attribute addProperty Size "142"}
{attribute addProperty Name "Term 11 (EK1100)"}
TYPE Term_11_EK1100_B6553301 EXTENDS EK1100_1FC0878B :
STRUCT
	{attribute addProperty Name "Term 12 (EL3174-0002)"}
	{attribute addProperty PreviousPort "Term 11 (EK1100) : B"}
	{attribute addProperty SyncUnit "Row_1"}
	Term_12_EL3174_0002 : EL3174_B71BFF42;
	{attribute addProperty Name "Term 13 (EL6001)"}
	{attribute addProperty PreviousPort "Term 12 (EL3174-0002) : B"}
	{attribute addProperty SyncUnit "Row_1"}
	Term_13_EL6001 : EL6001_0DE01E7E;
	{attribute addProperty Name "Term 14 (EL3011)"}
	{attribute addProperty PreviousPort "Term 13 (EL6001) : B"}
	{attribute addProperty SyncUnit "Row_1"}
	Term_14_EL3011 : EL3011_7A495228;
	{attribute addProperty Name "Term 15 (EL2008)"}
	{attribute addProperty PreviousPort "Term 14 (EL3011) : B"}
	{attribute addProperty SyncUnit "Row_1"}
	Term_15_EL2008 : EL2008_E2806B95;
	{attribute addProperty Name "Term 16 (EL2008)"}
	{attribute addProperty PreviousPort "Term 15 (EL2008) : B"}
	{attribute addProperty SyncUnit "Row_1"}
	Term_16_EL2008 : EL2008_E2806B95;
	{attribute addProperty Name "Term 17 (EK1110)"}
	{attribute addProperty PreviousPort "Term 16 (EL2008) : B"}
	{attribute addProperty SyncUnit "default"}
	Term_17_EK1110 : EK1110_1FC0878B;
END_STRUCT
END_TYPE

// ---- DUTs/IO/Topology/Term_18_EK1100_20659A8D.TcDUT
{attribute 'GeneratedUsingTerminal: EK1100-0000-0018'}
{attribute addProperty BoxType "EK1100-0000-0018"}
{attribute addProperty Id "Term_19_EL1809EL1809_32157CFD20Term_20_EL2809EL2809_2B6483BD19Term_21_EL1809EL1809_32157CFD20Term_22_EL3011EL3011_7A49522813Term_29_EL9011EL9011_D65D3D320"}
{attribute addProperty CRC "543529613"}
{attribute addProperty Size "72"}
{attribute addProperty Name "Term 18 (EK1100)"}
TYPE Term_18_EK1100_20659A8D EXTENDS EK1100_1FC0878B :
STRUCT
	{attribute addProperty Name "Term 19 (EL1809)"}
	{attribute addProperty PreviousPort "Term 18 (EK1100) : B"}
	{attribute addProperty SyncUnit "Row_1"}
	Term_19_EL1809 : EL1809_32157CFD;
	{attribute addProperty Name "Term 20 (EL2809)"}
	{attribute addProperty PreviousPort "Term 19 (EL1809) : B"}
	{attribute addProperty SyncUnit "Row_1"}
	Term_20_EL2809 : EL2809_2B6483BD;
	{attribute addProperty Name "Term 21 (EL1809)"}
	{attribute addProperty PreviousPort "Term 20 (EL2809) : B"}
	{attribute addProperty SyncUnit "Row_1"}
	Term_21_EL1809 : EL1809_32157CFD;
	{attribute addProperty Name "Term 22 (EL3011)"}
	{attribute addProperty PreviousPort "Term 21 (EL1809) : B"}
	{attribute addProperty SyncUnit "Row_1"}
	Term_22_EL3011 : EL3011_7A495228;
	{attribute addProperty Name "Term 29 (EL9011)"}
	{attribute addProperty PreviousPort "Term 22 (EL3011) : B"}
	{attribute addProperty SyncUnit "default"}
	Term_29_EL9011 : EL9011_D65D3D32;
END_STRUCT
END_TYPE

// ---- DUTs/IO/Topology/Term_25_EK1100_08217EB4.TcDUT
{attribute 'GeneratedUsingTerminal: EK1100-0000-0018'}
{attribute addProperty BoxType "EK1100-0000-0018"}
{attribute addProperty Id "Term_26_EL1819EL1819_32157CFD20Term_27_EL1819EL1819_32157CFD20Term_30_EL9011EL9011_D65D3D320"}
{attribute addProperty CRC "136412852"}
{attribute addProperty Size "40"}
{attribute addProperty Name "Term 25 (EK1100)"}
TYPE Term_25_EK1100_08217EB4 EXTENDS EK1100_1FC0878B :
STRUCT
	{attribute addProperty Name "Term 26 (EL1819)"}
	{attribute addProperty PreviousPort "Term 25 (EK1100) : B"}
	{attribute addProperty SyncUnit "Row_3"}
	Term_26_EL1819 : EL1819_32157CFD;
	{attribute addProperty Name "Term 27 (EL1819)"}
	{attribute addProperty PreviousPort "Term 26 (EL1819) : B"}
	{attribute addProperty SyncUnit "Row_3"}
	Term_27_EL1819 : EL1819_32157CFD;
	{attribute addProperty Name "Term 30 (EL9011)"}
	{attribute addProperty PreviousPort "Term 27 (EL1819) : B"}
	{attribute addProperty SyncUnit "default"}
	Term_30_EL9011 : EL9011_D65D3D32;
END_STRUCT
END_TYPE

// ---- DUTs/IO/Topology/Term_28_EK1100_415F4A7E.TcDUT
{attribute 'GeneratedUsingTerminal: EK1100-0000-0018'}
{attribute addProperty BoxType "EK1100-0000-0018"}
{attribute addProperty Id "Term_29_EL2788EL2788_E2806B9511Term_30_EL3773EL3773_F128CC82184Term_31_EL9011EL9011_D65D3D320"}
{attribute addProperty CRC "1096764030"}
{attribute addProperty Size "195"}
{attribute addProperty Name "Term 28 (EK1100)"}
TYPE Term_28_EK1100_415F4A7E EXTENDS EK1100_1FC0878B :
STRUCT
	{attribute addProperty Name "Term 29 (EL2788)"}
	{attribute addProperty PreviousPort "Term 28 (EK1100) : B"}
	{attribute addProperty SyncUnit "Row_4"}
	Term_29_EL2788 : EL2788_E2806B95;
	{attribute addProperty Name "Term 30 (EL3773)"}
	{attribute addProperty PreviousPort "Term 29 (EL2788) : B"}
	{attribute addProperty SyncUnit "Row_4"}
	Term_30_EL3773 : EL3773_F128CC82;
	{attribute addProperty Name "Term 31 (EL9011)"}
	{attribute addProperty PreviousPort "Term 30 (EL3773) : B"}
	{attribute addProperty SyncUnit "default"}
	Term_31_EL9011 : EL9011_D65D3D32;
END_STRUCT
END_TYPE

// ---- DUTs/IO/Topology/Term_24_EK1122_39E7B5CB.TcDUT
{attribute 'GeneratedUsingTerminal: EK1122-0000-0018'}
{attribute addProperty BoxType "EK1122-0000-0018"}
{attribute addProperty Id "Term_25_EK1100Term_25_EK1100_08217EB440Term_28_EK1100Term_28_EK1100_415F4A7E195"}
{attribute addProperty CRC "971486667"}
{attribute addProperty Size "235"}
{attribute addProperty Name "Term 24 (EK1122)"}
TYPE Term_24_EK1122_39E7B5CB EXTENDS EK1122_1FC0878B :
STRUCT
	{attribute addProperty Name "Term 25 (EK1100)"}
	{attribute addProperty PreviousPort "Term 24 (EK1122) : B"}
	{attribute addProperty SyncUnit "default"}
	Term_25_EK1100 : Term_25_EK1100_08217EB4;
	{attribute addProperty Name "Term 28 (EK1100)"}
	{attribute addProperty PreviousPort "Term 25 (EK1100) : C"}
	{attribute addProperty SyncUnit "default"}
	Term_28_EK1100 : Term_28_EK1100_415F4A7E;
END_STRUCT
END_TYPE

// ---- DUTs/IO/Topology/Term_23_EK1100_C1096874.TcDUT
{attribute 'GeneratedUsingTerminal: EK1100-0000-0018'}
{attribute addProperty BoxType "EK1100-0000-0018"}
{attribute addProperty Id "Term_24_EK1122Term_24_EK1122_39E7B5CB235Term_31_EL3773EL3773_F128CC82184Term_32_EL2258EL2258_E3B260FA508Term_33_EL3164EL3164_B71BFF4244Term_40_EK1110EK1110_1FC0878B2"}
{attribute addProperty CRC "3238619252"}
{attribute addProperty Size "973"}
{attribute addProperty Name "Term 23 (EK1100)"}
TYPE Term_23_EK1100_C1096874 EXTENDS EK1100_1FC0878B :
STRUCT
	{attribute addProperty Name "Term 24 (EK1122)"}
	{attribute addProperty PreviousPort "Term 23 (EK1100) : B"}
	{attribute addProperty SyncUnit "default"}
	Term_24_EK1122 : Term_24_EK1122_39E7B5CB;
	{attribute addProperty Name "Term 31 (EL3773)"}
	{attribute addProperty PreviousPort "Term 24 (EK1122) : C"}
	{attribute addProperty SyncUnit "Row_2"}
	Term_31_EL3773 : EL3773_F128CC82;
	{attribute addProperty Name "Term 32 (EL2258)"}
	{attribute addProperty PreviousPort "Term 31 (EL3773) : B"}
	{attribute addProperty SyncUnit "Row_2"}
	Term_32_EL2258 : EL2258_E3B260FA;
	{attribute addProperty Name "Term 33 (EL3164)"}
	{attribute addProperty PreviousPort "Term 32 (EL2258) : B"}
	{attribute addProperty SyncUnit "Row_2"}
	Term_33_EL3164 : EL3164_B71BFF42;
	{attribute addProperty Name "Term 40 (EK1110)"}
	{attribute addProperty PreviousPort "Term 33 (EL3164) : B"}
	{attribute addProperty SyncUnit "default"}
	Term_40_EK1110 : EK1110_1FC0878B;
END_STRUCT
END_TYPE

// ---- DUTs/IO/Topology/Term_42_EK1100_1039F2C4.TcDUT
{attribute 'GeneratedUsingTerminal: EK1100-0000-0018'}
{attribute addProperty BoxType "EK1100-0000-0018"}
{attribute addProperty Id "Term_43_EL1008EL1008_78E8D3DD12Term_44_EL1008EL1008_78E8D3DD12"}
{attribute addProperty CRC "272233156"}
{attribute addProperty Size "24"}
{attribute addProperty Name "Term 42 (EK1100)"}
TYPE Term_42_EK1100_1039F2C4 EXTENDS EK1100_1FC0878B :
STRUCT
	{attribute addProperty Name "Term 43 (EL1008)"}
	{attribute addProperty PreviousPort "Term 42 (EK1100) : B"}
	{attribute addProperty SyncUnit "default"}
	Term_43_EL1008 : EL1008_78E8D3DD;
	{attribute addProperty Name "Term 44 (EL1008)"}
	{attribute addProperty PreviousPort "Term 43 (EL1008) : B"}
	{attribute addProperty SyncUnit "default"}
	Term_44_EL1008 : EL1008_78E8D3DD;
END_STRUCT
END_TYPE

// ---- DUTs/IO/Topology/Term_10_EK1122_152EB6C2.TcDUT
{attribute 'GeneratedUsingTerminal: EK1122-0000-0018'}
{attribute addProperty BoxType "EK1122-0000-0018"}
{attribute addProperty Id "Term_11_EK1100Term_11_EK1100_B6553301142Term_18_EK1100Term_18_EK1100_20659A8D72Term_23_EK1100Term_23_EK1100_C1096874973Term_42_EK1100Term_42_EK1100_1039F2C424"}
{attribute addProperty CRC "355382978"}
{attribute addProperty Size "1211"}
{attribute addProperty Name "Term 10 (EK1122)"}
TYPE Term_10_EK1122_152EB6C2 EXTENDS EK1122_1FC0878B :
STRUCT
	{attribute addProperty Name "Term 11 (EK1100)"}
	{attribute addProperty PreviousPort "Term 10 (EK1122) : D"}
	{attribute addProperty SyncUnit "default"}
	Term_11_EK1100 : Term_11_EK1100_B6553301;
	{attribute addProperty Name "Term 18 (EK1100)"}
	{attribute addProperty PreviousPort "Term 17 (EK1110) : B"}
	{attribute addProperty SyncUnit "default"}
	Term_18_EK1100 : Term_18_EK1100_20659A8D;
	{attribute addProperty Name "Term 23 (EK1100)"}
	{attribute addProperty PreviousPort "Term 10 (EK1122) : B"}
	{attribute addProperty SyncUnit "default"}
	Term_23_EK1100 : Term_23_EK1100_C1096874;
	{attribute addProperty Name "Term 42 (EK1100)"}
	{attribute addProperty PreviousPort "Term 40 (EK1110) : B"}
	{attribute addProperty SyncUnit "default"}
	Term_42_EK1100 : Term_42_EK1100_1039F2C4;
END_STRUCT
END_TYPE

// ---- DUTs/IO/Topology/Term_9_EK1100_0DC40061.TcDUT
{attribute 'GeneratedUsingTerminal: EK1100-0000-0018'}
{attribute addProperty BoxType "EK1100-0000-0018"}
{attribute addProperty Id "Term_10_EK1122Term_10_EK1122_152EB6C21211Term_34_EL3403EL3403_812980A665Term_35_EL6001EL6001_0DE01E7E61Term_36_EL3024EL3024_C6E76B5A40Term_33_EL9011EL9011_D65D3D320"}
{attribute addProperty CRC "230948961"}
{attribute addProperty Size "1377"}
{attribute addProperty Name "Term 9 (EK1100)"}
TYPE Term_9_EK1100_0DC40061 EXTENDS EK1100_1FC0878B :
STRUCT
	{attribute addProperty Name "Term 10 (EK1122)"}
	{attribute addProperty PreviousPort "Term 9 (EK1100) : B"}
	{attribute addProperty SyncUnit "default"}
	Term_10_EK1122 : Term_10_EK1122_152EB6C2;
	{attribute addProperty Name "Term 34 (EL3403)"}
	{attribute addProperty PreviousPort "Term 10 (EK1122) : C"}
	{attribute addProperty SyncUnit "Row_0"}
	Term_34_EL3403 : EL3403_812980A6;
	{attribute addProperty Name "Term 35 (EL6001)"}
	{attribute addProperty PreviousPort "Term 34 (EL3403) : B"}
	{attribute addProperty SyncUnit "Row_0"}
	Term_35_EL6001 : EL6001_0DE01E7E;
	{attribute addProperty Name "Term 36 (EL3024)"}
	{attribute addProperty PreviousPort "Term 35 (EL6001) : B"}
	{attribute addProperty SyncUnit "Row_0"}
	Term_36_EL3024 : EL3024_C6E76B5A;
	{attribute addProperty Name "Term 33 (EL9011)"}
	{attribute addProperty PreviousPort "Term 36 (EL3024) : B"}
	{attribute addProperty SyncUnit "default"}
	Term_33_EL9011 : EL9011_D65D3D32;
END_STRUCT
END_TYPE

// ---- DUTs/IO/Topology/Device_2_EtherCAT_CA128DDC.TcDUT
{attribute 'GeneratedUsingTerminal: IODEVICETYPE_ETHERCATPROT'}
{attribute addProperty BoxType "IODEVICETYPE_ETHERCATPROT"}
{attribute addProperty Id "Term_9_EK1100Term_9_EK1100_0DC400611377SyncUnitsSyncUnits_91A42BBF108InputsInputs_A65FACA410OutputsOutputs_23C0ED1D6InfoDataInfoData_84133AC922"}
{attribute addProperty CRC "3390213596"}
{attribute addProperty Size "1523"}
{attribute addProperty Name "Device 2 (EtherCAT)"}
TYPE Device_2_EtherCAT_CA128DDC EXTENDS TcoIo.EtcMasterBase_62654B43 :
STRUCT
	{attribute addProperty Name "Term 9 (EK1100)"}
	{attribute addProperty PreviousPort "Device 2 (EtherCAT) : Master"}
	{attribute addProperty SyncUnit "default"}
	Term_9_EK1100 : Term_9_EK1100_0DC40061;
	{attribute addProperty Name "SyncUnits"}
	SyncUnits : SyncUnits_91A42BBF;
	{attribute addProperty Name "Inputs"}
	Inputs : TcoIo.Inputs_A65FACA4;
	{attribute addProperty Name "Outputs"}
	Outputs : TcoIo.Outputs_23C0ED1D;
	{attribute addProperty Name "InfoData"}
	InfoData : TcoIo.InfoData_84133AC9;
END_STRUCT
END_TYPE

// ---- DUTs/IO/Topology/Term_157_EK1100_7C4BDD77.TcDUT
{attribute 'GeneratedUsingTerminal: EK1100-0000-0018'}
{attribute addProperty BoxType "EK1100-0000-0018"}
{attribute addProperty Id "Term_159_EL1809EL1809_32157CFD20"}
{attribute addProperty CRC "2085346679"}
{attribute addProperty Size "20"}
{attribute addProperty Name "Term 157 (EK1100)"}
TYPE Term_157_EK1100_7C4BDD77 EXTENDS EK1100_1FC0878B :
STRUCT
	{attribute addProperty Name "Term 159 (EL1809)"}
	{attribute addProperty PreviousPort "Term 157 (EK1100) : B"}
	{attribute addProperty SyncUnit "default"}
	Term_159_EL1809 : EL1809_32157CFD;
END_STRUCT
END_TYPE

// ---- DUTs/IO/Topology/Term_158_EK1100_E3D699B1.TcDUT
{attribute 'GeneratedUsingTerminal: EK1100-0000-0018'}
{attribute addProperty BoxType "EK1100-0000-0018"}
{attribute addProperty Id "Term_160_EL1809EL1809_32157CFD20"}
{attribute addProperty CRC "3822492081"}
{attribute addProperty Size "20"}
{attribute addProperty Name "Term 158 (EK1100)"}
TYPE Term_158_EK1100_E3D699B1 EXTENDS EK1100_1FC0878B :
STRUCT
	{attribute addProperty Name "Term 160 (EL1809)"}
	{attribute addProperty PreviousPort "Term 158 (EK1100) : B"}
	{attribute addProperty SyncUnit "default"}
	Term_160_EL1809 : EL1809_32157CFD;
END_STRUCT
END_TYPE

// ---- DUTs/IO/Topology/Term_154_EK1122_E57516AE.TcDUT
{attribute 'GeneratedUsingTerminal: EK1122-0000-0018'}
{attribute addProperty BoxType "EK1122-0000-0018"}
{attribute addProperty Id "Term_157_EK1100Term_157_EK1100_7C4BDD7720Term_158_EK1100Term_158_EK1100_E3D699B120"}
{attribute addProperty CRC "3849655982"}
{attribute addProperty Size "40"}
{attribute addProperty Name "Term 154 (EK1122)"}
TYPE Term_154_EK1122_E57516AE EXTENDS EK1122_1FC0878B :
STRUCT
	{attribute addProperty Name "Term 157 (EK1100)"}
	{attribute addProperty PreviousPort "Term 154 (EK1122) : D"}
	{attribute addProperty SyncUnit "default"}
	Term_157_EK1100 : Term_157_EK1100_7C4BDD77;
	{attribute addProperty Name "Term 158 (EK1100)"}
	{attribute addProperty PreviousPort "Term 154 (EK1122) : B"}
	{attribute addProperty SyncUnit "default"}
	Term_158_EK1100 : Term_158_EK1100_E3D699B1;
END_STRUCT
END_TYPE

// ---- DUTs/IO/Topology/Term_153_EK1100_91C0BB48.TcDUT
{attribute 'GeneratedUsingTerminal: EK1100-0000-0018'}
{attribute addProperty BoxType "EK1100-0000-0018"}
{attribute addProperty Id "Term_154_EK1122Term_154_EK1122_E57516AE40Term_155_EL2008EL2008_E2806B9511Term_156_EL2008EL2008_E2806B9511"}
{attribute addProperty CRC "2445327176"}
{attribute addProperty Size "62"}
{attribute addProperty Name "Term 153 (EK1100)"}
TYPE Term_153_EK1100_91C0BB48 EXTENDS EK1100_1FC0878B :
STRUCT
	{attribute addProperty Name "Term 154 (EK1122)"}
	{attribute addProperty PreviousPort "Term 153 (EK1100) : B"}
	{attribute addProperty SyncUnit "default"}
	Term_154_EK1122 : Term_154_EK1122_E57516AE;
	{attribute addProperty Name "Term 155 (EL2008)"}
	{attribute addProperty PreviousPort "Term 154 (EK1122) : C"}
	{attribute addProperty SyncUnit "default"}
	Term_155_EL2008 : EL2008_E2806B95;
	{attribute addProperty Name "Term 156 (EL2008)"}
	{attribute addProperty PreviousPort "Term 155 (EL2008) : B"}
	{attribute addProperty SyncUnit "default"}
	Term_156_EL2008 : EL2008_E2806B95;
END_STRUCT
END_TYPE

// ---- DUTs/IO/Topology/Term_180_EK1100_796B7783.TcDUT
{attribute 'GeneratedUsingTerminal: EK1100-0000-0018'}
{attribute addProperty BoxType "EK1100-0000-0018"}
{attribute addProperty Id "Term_181_EL1809EL1809_32157CFD20"}
{attribute addProperty CRC "2037086083"}
{attribute addProperty Size "20"}
{attribute addProperty Name "Term 180 (EK1100)"}
TYPE Term_180_EK1100_796B7783 EXTENDS EK1100_1FC0878B :
STRUCT
	{attribute addProperty Name "Term 181 (EL1809)"}
	{attribute addProperty PreviousPort "Term 180 (EK1100) : B"}
	{attribute addProperty SyncUnit "default"}
	Term_181_EL1809 : EL1809_32157CFD;
END_STRUCT
END_TYPE

// ---- DUTs/IO/Topology/Term_182_EK1100_E6B2C35E.TcDUT
{attribute 'GeneratedUsingTerminal: EK1100-0000-0018'}
{attribute addProperty BoxType "EK1100-0000-0018"}
{attribute addProperty Id "Term_183_EL1809EL1809_32157CFD20"}
{attribute addProperty CRC "3870475102"}
{attribute addProperty Size "20"}
{attribute addProperty Name "Term 182 (EK1100)"}
TYPE Term_182_EK1100_E6B2C35E EXTENDS EK1100_1FC0878B :
STRUCT
	{attribute addProperty Name "Term 183 (EL1809)"}
	{attribute addProperty PreviousPort "Term 182 (EK1100) : B"}
	{attribute addProperty SyncUnit "default"}
	Term_183_EL1809 : EL1809_32157CFD;
END_STRUCT
END_TYPE

// ---- DUTs/IO/Topology/Term_179_EK1122_2A33725A.TcDUT
{attribute 'GeneratedUsingTerminal: EK1122-0000-0018'}
{attribute addProperty BoxType "EK1122-0000-0018"}
{attribute addProperty Id "Term_180_EK1100Term_180_EK1100_796B778320Term_182_EK1100Term_182_EK1100_E6B2C35E20"}
{attribute addProperty CRC "708014682"}
{attribute addProperty Size "40"}
{attribute addProperty Name "Term 179 (EK1122)"}
TYPE Term_179_EK1122_2A33725A EXTENDS EK1122_1FC0878B :
STRUCT
	{attribute addProperty Name "Term 180 (EK1100)"}
	{attribute addProperty PreviousPort "Term 179 (EK1122) : D"}
	{attribute addProperty SyncUnit "default"}
	Term_180_EK1100 : Term_180_EK1100_796B7783;
	{attribute addProperty Name "Term 182 (EK1100)"}
	{attribute addProperty PreviousPort "Term 179 (EK1122) : B"}
	{attribute addProperty SyncUnit "default"}
	Term_182_EK1100 : Term_182_EK1100_E6B2C35E;
END_STRUCT
END_TYPE

// ---- DUTs/IO/Topology/Term_178_EK1100_9B7E9852.TcDUT
{attribute 'GeneratedUsingTerminal: EK1100-0000-0018'}
{attribute addProperty BoxType "EK1100-0000-0018"}
{attribute addProperty Id "Term_179_EK1122Term_179_EK1122_2A33725A40Term_184_EL2008EL2008_E2806B9511Term_185_EL2008EL2008_E2806B9511"}
{attribute addProperty CRC "2608765010"}
{attribute addProperty Size "62"}
{attribute addProperty Name "Term 178 (EK1100)"}
TYPE Term_178_EK1100_9B7E9852 EXTENDS EK1100_1FC0878B :
STRUCT
	{attribute addProperty Name "Term 179 (EK1122)"}
	{attribute addProperty PreviousPort "Term 178 (EK1100) : B"}
	{attribute addProperty SyncUnit "default"}
	Term_179_EK1122 : Term_179_EK1122_2A33725A;
	{attribute addProperty Name "Term 184 (EL2008)"}
	{attribute addProperty PreviousPort "Term 179 (EK1122) : C"}
	{attribute addProperty SyncUnit "default"}
	Term_184_EL2008 : EL2008_E2806B95;
	{attribute addProperty Name "Term 185 (EL2008)"}
	{attribute addProperty PreviousPort "Term 184 (EL2008) : B"}
	{attribute addProperty SyncUnit "default"}
	Term_185_EL2008 : EL2008_E2806B95;
END_STRUCT
END_TYPE

// ---- DUTs/IO/Topology/Term_147_EK1122_CA6A5D16.TcDUT
{attribute 'GeneratedUsingTerminal: EK1122-0000-0018'}
{attribute addProperty BoxType "EK1122-0000-0018"}
{attribute addProperty Id "Term_153_EK1100Term_153_EK1100_91C0BB4862Term_178_EK1100Term_178_EK1100_9B7E985262"}
{attribute addProperty CRC "3395968278"}
{attribute addProperty Size "124"}
{attribute addProperty Name "Term 147 (EK1122)"}
TYPE Term_147_EK1122_CA6A5D16 EXTENDS EK1122_1FC0878B :
STRUCT
	{attribute addProperty Name "Term 153 (EK1100)"}
	{attribute addProperty PreviousPort "Term 147 (EK1122) : D"}
	{attribute addProperty SyncUnit "default"}
	Term_153_EK1100 : Term_153_EK1100_91C0BB48;
	{attribute addProperty Name "Term 178 (EK1100)"}
	{attribute addProperty PreviousPort "Term 147 (EK1122) : B"}
	{attribute addProperty SyncUnit "default"}
	Term_178_EK1100 : Term_178_EK1100_9B7E9852;
END_STRUCT
END_TYPE

// ---- DUTs/IO/Topology/Term_189_EK1100_06A16014.TcDUT
{attribute 'GeneratedUsingTerminal: EK1100-0000-0018'}
{attribute addProperty BoxType "EK1100-0000-0018"}
{attribute addProperty Id "Term_193_EL1809EL1809_32157CFD20"}
{attribute addProperty CRC "111239188"}
{attribute addProperty Size "20"}
{attribute addProperty Name "Term 189 (EK1100)"}
TYPE Term_189_EK1100_06A16014 EXTENDS EK1100_1FC0878B :
STRUCT
	{attribute addProperty Name "Term 193 (EL1809)"}
	{attribute addProperty PreviousPort "Term 189 (EK1100) : B"}
	{attribute addProperty SyncUnit "default"}
	Term_193_EL1809 : EL1809_32157CFD;
END_STRUCT
END_TYPE

// ---- DUTs/IO/Topology/Term_194_EK1100_D4E2C05F.TcDUT
{attribute 'GeneratedUsingTerminal: EK1100-0000-0018'}
{attribute addProperty BoxType "EK1100-0000-0018"}
{attribute addProperty Id "Term_200_EL1809EL1809_32157CFD20"}
{attribute addProperty CRC "3571630175"}
{attribute addProperty Size "20"}
{attribute addProperty Name "Term 194 (EK1100)"}
TYPE Term_194_EK1100_D4E2C05F EXTENDS EK1100_1FC0878B :
STRUCT
	{attribute addProperty Name "Term 200 (EL1809)"}
	{attribute addProperty PreviousPort "Term 194 (EK1100) : B"}
	{attribute addProperty SyncUnit "default"}
	Term_200_EL1809 : EL1809_32157CFD;
END_STRUCT
END_TYPE

// ---- DUTs/IO/Topology/Term_188_EK1122_78D8AA43.TcDUT
{attribute 'GeneratedUsingTerminal: EK1122-0000-0018'}
{attribute addProperty BoxType "EK1122-0000-0018"}
{attribute addProperty Id "Term_189_EK1100Term_189_EK1100_06A1601420Term_194_EK1100Term_194_EK1100_D4E2C05F20"}
{attribute addProperty CRC "2027465283"}
{attribute addProperty Size "40"}
{attribute addProperty Name "Term 188 (EK1122)"}
TYPE Term_188_EK1122_78D8AA43 EXTENDS EK1122_1FC0878B :
STRUCT
	{attribute addProperty Name "Term 189 (EK1100)"}
	{attribute addProperty PreviousPort "Term 188 (EK1122) : D"}
	{attribute addProperty SyncUnit "default"}
	Term_189_EK1100 : Term_189_EK1100_06A16014;
	{attribute addProperty Name "Term 194 (EK1100)"}
	{attribute addProperty PreviousPort "Term 188 (EK1122) : B"}
	{attribute addProperty SyncUnit "default"}
	Term_194_EK1100 : Term_194_EK1100_D4E2C05F;
END_STRUCT
END_TYPE

// ---- DUTs/IO/Topology/Term_187_EK1100_648C31BD.TcDUT
{attribute 'GeneratedUsingTerminal: EK1100-0000-0018'}
{attribute addProperty BoxType "EK1100-0000-0018"}
{attribute addProperty Id "Term_188_EK1122Term_188_EK1122_78D8AA4340Term_204_EL2008EL2008_E2806B9511Term_205_EL2008EL2008_E2806B9511"}
{attribute addProperty CRC "1686909373"}
{attribute addProperty Size "62"}
{attribute addProperty Name "Term 187 (EK1100)"}
TYPE Term_187_EK1100_648C31BD EXTENDS EK1100_1FC0878B :
STRUCT
	{attribute addProperty Name "Term 188 (EK1122)"}
	{attribute addProperty PreviousPort "Term 187 (EK1100) : B"}
	{attribute addProperty SyncUnit "default"}
	Term_188_EK1122 : Term_188_EK1122_78D8AA43;
	{attribute addProperty Name "Term 204 (EL2008)"}
	{attribute addProperty PreviousPort "Term 188 (EK1122) : C"}
	{attribute addProperty SyncUnit "default"}
	Term_204_EL2008 : EL2008_E2806B95;
	{attribute addProperty Name "Term 205 (EL2008)"}
	{attribute addProperty PreviousPort "Term 204 (EL2008) : B"}
	{attribute addProperty SyncUnit "default"}
	Term_205_EL2008 : EL2008_E2806B95;
END_STRUCT
END_TYPE

// ---- DUTs/IO/Topology/Term_231_EK1100_6FCE8CEB.TcDUT
{attribute 'GeneratedUsingTerminal: EK1100-0000-0018'}
{attribute addProperty BoxType "EK1100-0000-0018"}
{attribute addProperty Id "Term_232_EL1809EL1809_32157CFD20"}
{attribute addProperty CRC "1875807467"}
{attribute addProperty Size "20"}
{attribute addProperty Name "Term 231 (EK1100)"}
TYPE Term_231_EK1100_6FCE8CEB EXTENDS EK1100_1FC0878B :
STRUCT
	{attribute addProperty Name "Term 232 (EL1809)"}
	{attribute addProperty PreviousPort "Term 231 (EK1100) : B"}
	{attribute addProperty SyncUnit "default"}
	Term_232_EL1809 : EL1809_32157CFD;
END_STRUCT
END_TYPE

// ---- DUTs/IO/Topology/Term_233_EK1100_CB654C3B.TcDUT
{attribute 'GeneratedUsingTerminal: EK1100-0000-0018'}
{attribute addProperty BoxType "EK1100-0000-0018"}
{attribute addProperty Id "Term_234_EL1809EL1809_32157CFD20"}
{attribute addProperty CRC "3412413499"}
{attribute addProperty Size "20"}
{attribute addProperty Name "Term 233 (EK1100)"}
TYPE Term_233_EK1100_CB654C3B EXTENDS EK1100_1FC0878B :
STRUCT
	{attribute addProperty Name "Term 234 (EL1809)"}
	{attribute addProperty PreviousPort "Term 233 (EK1100) : B"}
	{attribute addProperty SyncUnit "default"}
	Term_234_EL1809 : EL1809_32157CFD;
END_STRUCT
END_TYPE

// ---- DUTs/IO/Topology/Term_230_EK1122_16418046.TcDUT
{attribute 'GeneratedUsingTerminal: EK1122-0000-0018'}
{attribute addProperty BoxType "EK1122-0000-0018"}
{attribute addProperty Id "Term_231_EK1100Term_231_EK1100_6FCE8CEB20Term_233_EK1100Term_233_EK1100_CB654C3B20"}
{attribute addProperty CRC "373391430"}
{attribute addProperty Size "40"}
{attribute addProperty Name "Term 230 (EK1122)"}
TYPE Term_230_EK1122_16418046 EXTENDS EK1122_1FC0878B :
STRUCT
	{attribute addProperty Name "Term 231 (EK1100)"}
	{attribute addProperty PreviousPort "Term 230 (EK1122) : D"}
	{attribute addProperty SyncUnit "default"}
	Term_231_EK1100 : Term_231_EK1100_6FCE8CEB;
	{attribute addProperty Name "Term 233 (EK1100)"}
	{attribute addProperty PreviousPort "Term 230 (EK1122) : B"}
	{attribute addProperty SyncUnit "default"}
	Term_233_EK1100 : Term_233_EK1100_CB654C3B;
END_STRUCT
END_TYPE

// ---- DUTs/IO/Topology/Term_207_EK1100_2D36550A.TcDUT
{attribute 'GeneratedUsingTerminal: EK1100-0000-0018'}
{attribute addProperty BoxType "EK1100-0000-0018"}
{attribute addProperty Id "Term_230_EK1122Term_230_EK1122_1641804640Term_235_EL2008EL2008_E2806B9511Term_236_EL2008EL2008_E2806B9511"}
{attribute addProperty CRC "758535434"}
{attribute addProperty Size "62"}
{attribute addProperty Name "Term 207 (EK1100)"}
TYPE Term_207_EK1100_2D36550A EXTENDS EK1100_1FC0878B :
STRUCT
	{attribute addProperty Name "Term 230 (EK1122)"}
	{attribute addProperty PreviousPort "Term 207 (EK1100) : B"}
	{attribute addProperty SyncUnit "default"}
	Term_230_EK1122 : Term_230_EK1122_16418046;
	{attribute addProperty Name "Term 235 (EL2008)"}
	{attribute addProperty PreviousPort "Term 230 (EK1122) : C"}
	{attribute addProperty SyncUnit "default"}
	Term_235_EL2008 : EL2008_E2806B95;
	{attribute addProperty Name "Term 236 (EL2008)"}
	{attribute addProperty PreviousPort "Term 235 (EL2008) : B"}
	{attribute addProperty SyncUnit "default"}
	Term_236_EL2008 : EL2008_E2806B95;
END_STRUCT
END_TYPE

// ---- DUTs/IO/Topology/Term_186_EK1122_75C79D52.TcDUT
{attribute 'GeneratedUsingTerminal: EK1122-0000-0018'}
{attribute addProperty BoxType "EK1122-0000-0018"}
{attribute addProperty Id "Term_187_EK1100Term_187_EK1100_648C31BD62Term_207_EK1100Term_207_EK1100_2D36550A62"}
{attribute addProperty CRC "1976016210"}
{attribute addProperty Size "124"}
{attribute addProperty Name "Term 186 (EK1122)"}
TYPE Term_186_EK1122_75C79D52 EXTENDS EK1122_1FC0878B :
STRUCT
	{attribute addProperty Name "Term 187 (EK1100)"}
	{attribute addProperty PreviousPort "Term 186 (EK1122) : D"}
	{attribute addProperty SyncUnit "default"}
	Term_187_EK1100 : Term_187_EK1100_648C31BD;
	{attribute addProperty Name "Term 207 (EK1100)"}
	{attribute addProperty PreviousPort "Term 186 (EK1122) : B"}
	{attribute addProperty SyncUnit "default"}
	Term_207_EK1100 : Term_207_EK1100_2D36550A;
END_STRUCT
END_TYPE

// ---- DUTs/IO/Topology/Term_237_EK1122_86A8F7BD.TcDUT
{attribute 'GeneratedUsingTerminal: EK1122-0000-0018'}
{attribute addProperty BoxType "EK1122-0000-0018"}
{attribute addProperty Id "Drive_238_AX5101_0000_0214AX5101_1BD22F5129"}
{attribute addProperty CRC "2259220413"}
{attribute addProperty Size "29"}
{attribute addProperty Name "Term 237 (EK1122)"}
TYPE Term_237_EK1122_86A8F7BD EXTENDS EK1122_1FC0878B :
STRUCT
	{attribute addProperty Name "Drive 238 (AX5101-0000-0214)"}
	{attribute addProperty PreviousPort "Term 237 (EK1122) : D"}
	{attribute addProperty SyncUnit "default"}
	Drive_238_AX5101_0000_0214 : AX5101_1BD22F51;
END_STRUCT
END_TYPE

// ---- DUTs/IO/Topology/Term_289_EK1100_9C677E50.TcDUT
{attribute 'GeneratedUsingTerminal: EK1100-0000-0018'}
{attribute addProperty BoxType "EK1100-0000-0018"}
{attribute addProperty Id "Term_237_EK1122Term_237_EK1122_86A8F7BD29Term_293_EL1809EL1809_32157CFD20"}
{attribute addProperty CRC "2624028240"}
{attribute addProperty Size "49"}
{attribute addProperty Name "Term 289 (EK1100)"}
TYPE Term_289_EK1100_9C677E50 EXTENDS EK1100_1FC0878B :
STRUCT
	{attribute addProperty Name "Term 237 (EK1122)"}
	{attribute addProperty PreviousPort "Term 289 (EK1100) : B"}
	{attribute addProperty SyncUnit "default"}
	Term_237_EK1122 : Term_237_EK1122_86A8F7BD;
	{attribute addProperty Name "Term 293 (EL1809)"}
	{attribute addProperty PreviousPort "Term 237 (EK1122) : C"}
	{attribute addProperty SyncUnit "default"}
	Term_293_EL1809 : EL1809_32157CFD;
END_STRUCT
END_TYPE

// ---- DUTs/IO/Topology/Term_294_EK1100_DFE2A59E.TcDUT
{attribute 'GeneratedUsingTerminal: EK1100-0000-0018'}
{attribute addProperty BoxType "EK1100-0000-0018"}
{attribute addProperty Id "Term_300_EL1809EL1809_32157CFD20Term_304_EL2008EL2008_E2806B9511Term_305_EL2008EL2008_E2806B9511"}
{attribute addProperty CRC "3756172702"}
{attribute addProperty Size "42"}
{attribute addProperty Name "Term 294 (EK1100)"}
TYPE Term_294_EK1100_DFE2A59E EXTENDS EK1100_1FC0878B :
STRUCT
	{attribute addProperty Name "Term 300 (EL1809)"}
	{attribute addProperty PreviousPort "Term 294 (EK1100) : B"}
	{attribute addProperty SyncUnit "default"}
	Term_300_EL1809 : EL1809_32157CFD;
	{attribute addProperty Name "Term 304 (EL2008)"}
	{attribute addProperty PreviousPort "Term 300 (EL1809) : B"}
	{attribute addProperty SyncUnit "default"}
	Term_304_EL2008 : EL2008_E2806B95;
	{attribute addProperty Name "Term 305 (EL2008)"}
	{attribute addProperty PreviousPort "Term 304 (EL2008) : B"}
	{attribute addProperty SyncUnit "default"}
	Term_305_EL2008 : EL2008_E2806B95;
END_STRUCT
END_TYPE

// ---- DUTs/IO/Topology/Term_331_EK1100_B9C4E092.TcDUT
{attribute 'GeneratedUsingTerminal: EK1100-0000-0018'}
{attribute addProperty BoxType "EK1100-0000-0018"}
{attribute addProperty Id "Term_332_EL1809EL1809_32157CFD20"}
{attribute addProperty CRC "3116687506"}
{attribute addProperty Size "20"}
{attribute addProperty Name "Term 331 (EK1100)"}
TYPE Term_331_EK1100_B9C4E092 EXTENDS EK1100_1FC0878B :
STRUCT
	{attribute addProperty Name "Term 332 (EL1809)"}
	{attribute addProperty PreviousPort "Term 331 (EK1100) : B"}
	{attribute addProperty SyncUnit "default"}
	Term_332_EL1809 : EL1809_32157CFD;
END_STRUCT
END_TYPE

// ---- DUTs/IO/Topology/Term_333_EK1100_1D6F2042.TcDUT
{attribute 'GeneratedUsingTerminal: EK1100-0000-0018'}
{attribute addProperty BoxType "EK1100-0000-0018"}
{attribute addProperty Id "Term_334_EL1809EL1809_32157CFD20"}
{attribute addProperty CRC "493822018"}
{attribute addProperty Size "20"}
{attribute addProperty Name "Term 333 (EK1100)"}
TYPE Term_333_EK1100_1D6F2042 EXTENDS EK1100_1FC0878B :
STRUCT
	{attribute addProperty Name "Term 334 (EL1809)"}
	{attribute addProperty PreviousPort "Term 333 (EK1100) : B"}
	{attribute addProperty SyncUnit "default"}
	Term_334_EL1809 : EL1809_32157CFD;
END_STRUCT
END_TYPE

// ---- DUTs/IO/Topology/Term_330_EK1122_0EDE60FE.TcDUT
{attribute 'GeneratedUsingTerminal: EK1122-0000-0018'}
{attribute addProperty BoxType "EK1122-0000-0018"}
{attribute addProperty Id "Term_331_EK1100Term_331_EK1100_B9C4E09220Term_333_EK1100Term_333_EK1100_1D6F204220"}
{attribute addProperty CRC "249454846"}
{attribute addProperty Size "40"}
{attribute addProperty Name "Term 330 (EK1122)"}
TYPE Term_330_EK1122_0EDE60FE EXTENDS EK1122_1FC0878B :
STRUCT
	{attribute addProperty Name "Term 331 (EK1100)"}
	{attribute addProperty PreviousPort "Term 330 (EK1122) : D"}
	{attribute addProperty SyncUnit "default"}
	Term_331_EK1100 : Term_331_EK1100_B9C4E092;
	{attribute addProperty Name "Term 333 (EK1100)"}
	{attribute addProperty PreviousPort "Term 331 (EK1100) : C"}
	{attribute addProperty SyncUnit "default"}
	Term_333_EK1100 : Term_333_EK1100_1D6F2042;
END_STRUCT
END_TYPE

// ---- DUTs/IO/Topology/Term_307_EK1100_EB8FAA41.TcDUT
{attribute 'GeneratedUsingTerminal: EK1100-0000-0018'}
{attribute addProperty BoxType "EK1100-0000-0018"}
{attribute addProperty Id "Term_330_EK1122Term_330_EK1122_0EDE60FE40Term_335_EL2008EL2008_E2806B9511Term_336_EL2008EL2008_E2806B9511"}
{attribute addProperty CRC "3952060993"}
{attribute addProperty Size "62"}
{attribute addProperty Name "Term 307 (EK1100)"}
TYPE Term_307_EK1100_EB8FAA41 EXTENDS EK1100_1FC0878B :
STRUCT
	{attribute addProperty Name "Term 330 (EK1122)"}
	{attribute addProperty PreviousPort "Term 307 (EK1100) : B"}
	{attribute addProperty SyncUnit "default"}
	Term_330_EK1122 : Term_330_EK1122_0EDE60FE;
	{attribute addProperty Name "Term 335 (EL2008)"}
	{attribute addProperty PreviousPort "Term 330 (EK1122) : C"}
	{attribute addProperty SyncUnit "default"}
	Term_335_EL2008 : EL2008_E2806B95;
	{attribute addProperty Name "Term 336 (EL2008)"}
	{attribute addProperty PreviousPort "Term 335 (EL2008) : B"}
	{attribute addProperty SyncUnit "default"}
	Term_336_EL2008 : EL2008_E2806B95;
END_STRUCT
END_TYPE

// ---- DUTs/IO/Topology/Term_288_EK1122_18F8921F.TcDUT
{attribute 'GeneratedUsingTerminal: EK1122-0000-0018'}
{attribute addProperty BoxType "EK1122-0000-0018"}
{attribute addProperty Id "Term_289_EK1100Term_289_EK1100_9C677E5049Term_294_EK1100Term_294_EK1100_DFE2A59E42Term_307_EK1100Term_307_EK1100_EB8FAA4162"}
{attribute addProperty CRC "418943519"}
{attribute addProperty Size "153"}
{attribute addProperty Name "Term 288 (EK1122)"}
TYPE Term_288_EK1122_18F8921F EXTENDS EK1122_1FC0878B :
STRUCT
	{attribute addProperty Name "Term 289 (EK1100)"}
	{attribute addProperty PreviousPort "Term 288 (EK1122) : D"}
	{attribute addProperty SyncUnit "default"}
	Term_289_EK1100 : Term_289_EK1100_9C677E50;
	{attribute addProperty Name "Term 294 (EK1100)"}
	{attribute addProperty PreviousPort "Term 289 (EK1100) : C"}
	{attribute addProperty SyncUnit "default"}
	Term_294_EK1100 : Term_294_EK1100_DFE2A59E;
	{attribute addProperty Name "Term 307 (EK1100)"}
	{attribute addProperty PreviousPort "Term 294 (EK1100) : C"}
	{attribute addProperty SyncUnit "default"}
	Term_307_EK1100 : Term_307_EK1100_EB8FAA41;
END_STRUCT
END_TYPE

// ---- DUTs/IO/Topology/Term_146_EK1100_439F5464.TcDUT
{attribute 'GeneratedUsingTerminal: EK1100-0000-0018'}
{attribute addProperty BoxType "EK1100-0000-0018"}
{attribute addProperty Id "Term_147_EK1122Term_147_EK1122_CA6A5D16124Term_186_EK1122Term_186_EK1122_75C79D52124Term_148_EL1809EL1809_32157CFD20Term_149_EL1809EL1809_32157CFD20Term_150_EL1809EL1809_32157CFD20Term_151_EL1809EL1809_32157CFD20Term_152_EL1809EL1809_32157CFD20Term_288_EK1122Term_288_EK1122_18F8921F153Term_1158_EL2008EL2008_E2806B9511Term_1159_EL2008EL2008_E2806B9511Term_1160_EL2008EL2008_E2806B9511Term_1161_EL2008EL2008_E2806B9511Term_1162_EL2008EL2008_E2806B9511Term_1163_EL2008EL2008_E2806B9511"}
{attribute addProperty CRC "1134515300"}
{attribute addProperty Size "567"}
{attribute addProperty Name "Term 146 (EK1100)"}
TYPE Term_146_EK1100_439F5464 EXTENDS EK1100_1FC0878B :
STRUCT
	{attribute addProperty Name "Term 147 (EK1122)"}
	{attribute addProperty PreviousPort "Term 146 (EK1100) : B"}
	{attribute addProperty SyncUnit "default"}
	Term_147_EK1122 : Term_147_EK1122_CA6A5D16;
	{attribute addProperty Name "Term 186 (EK1122)"}
	{attribute addProperty PreviousPort "Term 147 (EK1122) : C"}
	{attribute addProperty SyncUnit "default"}
	Term_186_EK1122 : Term_186_EK1122_75C79D52;
	{attribute addProperty Name "Term 148 (EL1809)"}
	{attribute addProperty PreviousPort "Term 186 (EK1122) : C"}
	{attribute addProperty SyncUnit "default"}
	Term_148_EL1809 : EL1809_32157CFD;
	{attribute addProperty Name "Term 149 (EL1809)"}
	{attribute addProperty PreviousPort "Term 148 (EL1809) : B"}
	{attribute addProperty SyncUnit "default"}
	Term_149_EL1809 : EL1809_32157CFD;
	{attribute addProperty Name "Term 150 (EL1809)"}
	{attribute addProperty PreviousPort "Term 149 (EL1809) : B"}
	{attribute addProperty SyncUnit "default"}
	Term_150_EL1809 : EL1809_32157CFD;
	{attribute addProperty Name "Term 151 (EL1809)"}
	{attribute addProperty PreviousPort "Term 150 (EL1809) : B"}
	{attribute addProperty SyncUnit "default"}
	Term_151_EL1809 : EL1809_32157CFD;
	{attribute addProperty Name "Term 152 (EL1809)"}
	{attribute addProperty PreviousPort "Term 151 (EL1809) : B"}
	{attribute addProperty SyncUnit "default"}
	Term_152_EL1809 : EL1809_32157CFD;
	{attribute addProperty Name "Term 288 (EK1122)"}
	{attribute addProperty PreviousPort "Term 152 (EL1809) : B"}
	{attribute addProperty SyncUnit "default"}
	Term_288_EK1122 : Term_288_EK1122_18F8921F;
	{attribute addProperty Name "Term 1158 (EL2008)"}
	{attribute addProperty PreviousPort "Term 288 (EK1122) : C"}
	{attribute addProperty SyncUnit "default"}
	Term_1158_EL2008 : EL2008_E2806B95;
	{attribute addProperty Name "Term 1159 (EL2008)"}
	{attribute addProperty PreviousPort "Term 1158 (EL2008) : B"}
	{attribute addProperty SyncUnit "default"}
	Term_1159_EL2008 : EL2008_E2806B95;
	{attribute addProperty Name "Term 1160 (EL2008)"}
	{attribute addProperty PreviousPort "Term 1159 (EL2008) : B"}
	{attribute addProperty SyncUnit "default"}
	Term_1160_EL2008 : EL2008_E2806B95;
	{attribute addProperty Name "Term 1161 (EL2008)"}
	{attribute addProperty PreviousPort "Term 1160 (EL2008) : B"}
	{attribute addProperty SyncUnit "default"}
	Term_1161_EL2008 : EL2008_E2806B95;
	{attribute addProperty Name "Term 1162 (EL2008)"}
	{attribute addProperty PreviousPort "Term 1161 (EL2008) : B"}
	{attribute addProperty SyncUnit "default"}
	Term_1162_EL2008 : EL2008_E2806B95;
	{attribute addProperty Name "Term 1163 (EL2008)"}
	{attribute addProperty PreviousPort "Term 1162 (EL2008) : B"}
	{attribute addProperty SyncUnit "default"}
	Term_1163_EL2008 : EL2008_E2806B95;
END_STRUCT
END_TYPE

// ---- DUTs/IO/Topology/Device_3_EtherCAT_CA191EDE.TcDUT
{attribute 'GeneratedUsingTerminal: IODEVICETYPE_ETHERCATPROT'}
{attribute addProperty BoxType "IODEVICETYPE_ETHERCATPROT"}
{attribute addProperty Id "Term_146_EK1100Term_146_EK1100_439F5464567SyncUnitsSyncUnits_67D36DDA18InputsInputs_A65FACA410OutputsOutputs_23C0ED1D6InfoDataInfoData_84133AC922"}
{attribute addProperty CRC "3390643934"}
{attribute addProperty Size "623"}
{attribute addProperty Name "Device 3 (EtherCAT)"}
TYPE Device_3_EtherCAT_CA191EDE EXTENDS TcoIo.EtcMasterBase_62654B43 :
STRUCT
	{attribute addProperty Name "Term 146 (EK1100)"}
	{attribute addProperty PreviousPort "Device 3 (EtherCAT) : Master"}
	{attribute addProperty SyncUnit "default"}
	Term_146_EK1100 : Term_146_EK1100_439F5464;
	{attribute addProperty Name "SyncUnits"}
	SyncUnits : SyncUnits_67D36DDA;
	{attribute addProperty Name "Inputs"}
	Inputs : TcoIo.Inputs_A65FACA4;
	{attribute addProperty Name "Outputs"}
	Outputs : TcoIo.Outputs_23C0ED1D;
	{attribute addProperty Name "InfoData"}
	InfoData : TcoIo.InfoData_84133AC9;
END_STRUCT
END_TYPE

// ---- GVLs/GVL_iXlinker.TcGVL
{attribute 'qualified_only'}
VAR_GLOBAL
		Device_1_EtherCAT : Device_1_EtherCAT_B557D6C6;
		Device_2_EtherCAT : Device_2_EtherCAT_CA128DDC;
		Device_3_EtherCAT : Device_3_EtherCAT_CA191EDE;
END_VAR

// ---- POUs/MAIN.TcPOU
PROGRAM MAIN
VAR
END_VAR

END_PROGRAM
